// StandardPLC/Application/IO_CONFIG/INPUT_CONFIG_PI
PROGRAM INPUT_CONFIG_PI
VAR
	
	INPUT_A25: ifmFastInput.IncEncoder;
	CFDiag_INPUT_A25: ifmIOconfigDiagProt.ConfigDiagProt;
	INPUT_A26: ifmFastInput.IncEncoder;
	CFDiag_INPUT_A26: ifmIOconfigDiagProt.ConfigDiagProt;
	INPUT_A27: ifmFastInput.FastCount;
	CFDiag_INPUT_A27: ifmIOconfigDiagProt.ConfigDiagProt;
	INPUT_A28: ifmFastInput.FastCount;
	CFDiag_INPUT_A28: ifmIOconfigDiagProt.ConfigDiagProt;
	SET: ARRAY[0..70] OF SR;
	FastCount_0: ifmFastInput.FastCount;
	x1: BOOL;
	x2: REAL;
	x3: BOOL;
	x4: REAL;
END_VAR
VAR // added by the converter: edge detectors and wires of the graphical bodies
    _rt1, _rt2, _rt3, _rt4 : R_TRIG;
END_VAR

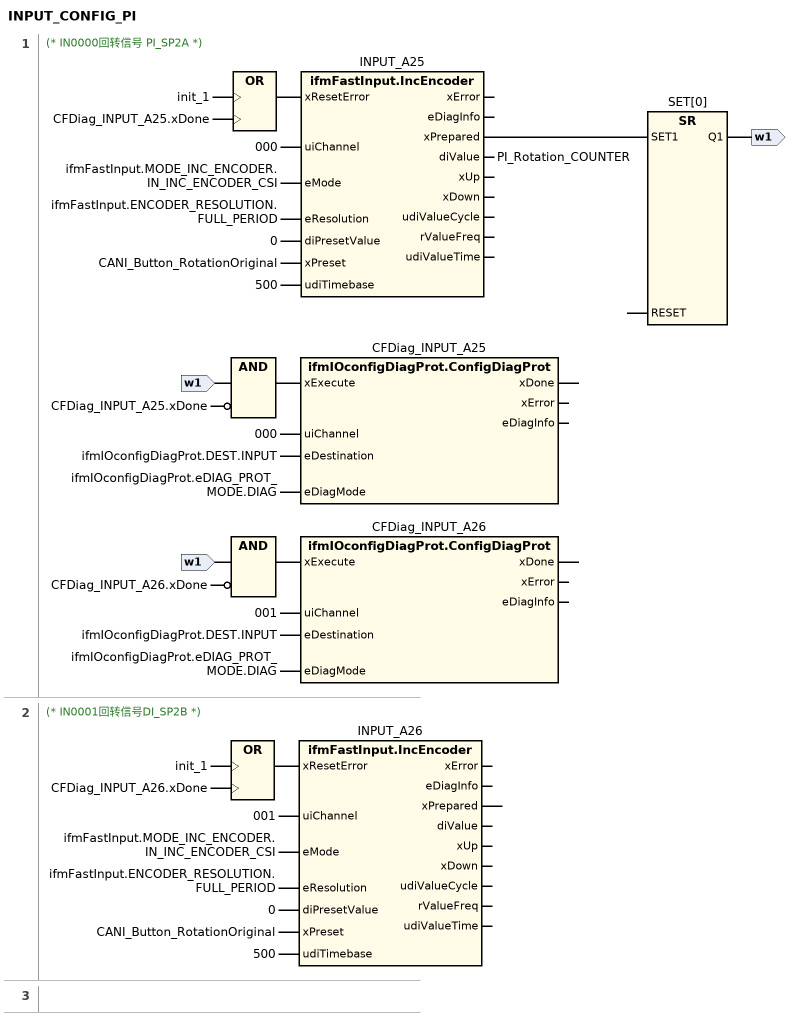
// NETWORK 1
//    (* IN0000回转信号 PI_SP2A *)
_rt1(CLK := init_1);
_rt2(CLK := CFDiag_INPUT_A25.xDone);
INPUT_A25(
    xResetError := _rt1.Q OR _rt2.Q,
    uiChannel := 000,
    eMode := ifmFastInput.MODE_INC_ENCODER.IN_INC_ENCODER_CSI,
    eResolution := ifmFastInput.ENCODER_RESOLUTION.FULL_PERIOD,
    diPresetValue := 0,
    xPreset := CANI_Button_RotationOriginal,
    udiTimebase := 500,
    diValue => PI_Rotation_COUNTER); // ifmFastInput.IncEncoder
SET[0](SET1 := INPUT_A25.xPrepared); // SR
CFDiag_INPUT_A25(
    xExecute := SET[0].Q1 AND NOT CFDiag_INPUT_A25.xDone,
    uiChannel := 000,
    eDestination := ifmIOconfigDiagProt.DEST.INPUT,
    eDiagMode := ifmIOconfigDiagProt.eDIAG_PROT_MODE.DIAG); // ifmIOconfigDiagProt.ConfigDiagProt
CFDiag_INPUT_A26(
    xExecute := SET[0].Q1 AND NOT CFDiag_INPUT_A26.xDone,
    uiChannel := 001,
    eDestination := ifmIOconfigDiagProt.DEST.INPUT,
    eDiagMode := ifmIOconfigDiagProt.eDIAG_PROT_MODE.DIAG); // ifmIOconfigDiagProt.ConfigDiagProt

// NETWORK 2
// (* IN0001回转信号DI_SP2B *)
_rt3(CLK := init_1);
_rt4(CLK := CFDiag_INPUT_A26.xDone);
INPUT_A26(
    xResetError := _rt3.Q OR _rt4.Q,
    uiChannel := 001,
    eMode := ifmFastInput.MODE_INC_ENCODER.IN_INC_ENCODER_CSI,
    eResolution := ifmFastInput.ENCODER_RESOLUTION.FULL_PERIOD,
    diPresetValue := 0,
    xPreset := CANI_Button_RotationOriginal,
    udiTimebase := 500); // ifmFastInput.IncEncoder

// NETWORK 3

END_PROGRAM

// StandardPLC/Application/IO_CONFIG/OUTPUT_CONFID
PROGRAM OUTPUT_CONFID
VAR
	SYSTEMSUPPLY:ifmIOcommon.SystemSupply;
	OUTGROUP0:ifmOutGroup.OutputGroup;
	OUTGROUP1:ifmOutGroup.OutputGroup;
	OUTGROUP2:ifmOutGroup.OutputGroup;
	OUTGROUP3:ifmOutGroup.OutputGroup;
	OUTGROUP4:ifmOutGroup.OutputGroup;
	OUTGROUP5:ifmOutGroup.OutputGroup;
(*******PWM*******)
	PWMI_A06: ifmOutPWM.CurrentControl;
//	PWMI_A06: ifmOutPWM.PWM1000;
	PWMI_A07: ifmOutPWM.PWM1000;
	PWMI_A08: ifmOutPWM.CurrentControl;
	PWMI_A09: ifmOutPWM.PWM1000;
	PWMI_A10: ifmOutPWM.CurrentControl;
	PWMI_A11: ifmOutPWM.PWM1000;
	PWMI_A12: ifmOutPWM.CurrentControl;
	PWMI_A13: ifmOutPWM.CurrentControl;
	PWMI_A14: ifmOutPWM.CurrentControl;
	PWMI_A16: ifmOutPWM.CurrentControl;
//	PWMI_A16: ifmOutPWM.PWM1000;
	PWMI_A17: ifmOutPWM.PWM1000;
	PWMI_A18: ifmOutPWM.CurrentControl;
//	PWMI_A18: CONTROL_OCC_CR7xxS;
	PWMI_A19: ifmOutPWM.PWM1000;
	PWMI_A20: ifmOutPWM.CurrentControl;
	PWMI_A21: ifmOutPWM.PWM1000;
	PWMI_A22: ifmOutPWM.CurrentControl;
	PWMI_A23: ifmOutPWM.CurrentControl;
	PWMI_A24: ifmOutPWM.CurrentControl;
	PWMI_A73: ifmOutPWM.CurrentControl;
	PWMI_A74: ifmOutPWM.PWM1000;
	PWMI_A75: ifmOutPWM.CurrentControl;
	PWMI_A76: ifmOutPWM.PWM1000;
	PWMI_A77: ifmOutPWM.CurrentControl;
	PWMI_A78: ifmOutPWM.PWM1000;
	PWMI_A79: ifmOutPWM.CurrentControl;
	PWMI_A80: ifmOutPWM.CurrentControl;
	PWMI_A81: ifmOutPWM.CurrentControl;
	
	PWMI_B16: ifmOutPWM.CurrentControl;
	PWMI_B17: ifmOutPWM.PWM1000;
	PWMI_B18: ifmOutPWM.CurrentControl;
	PWMI_B19: ifmOutPWM.PWM1000;
	PWMI_B20: ifmOutPWM.CurrentControl;
	PWMI_B21: ifmOutPWM.PWM1000;
	PWMI_B22: ifmOutPWM.CurrentControl;
	PWMI_B23: ifmOutPWM.CurrentControl;
	PWMI_B24: ifmOutPWM.CurrentControl;
	PWMI_B63: ifmOutPWM.CurrentControl;
	PWMI_B64: ifmOutPWM.PWM1000;
	PWMI_B65: ifmOutPWM.CurrentControl;
	PWMI_B66: ifmOutPWM.PWM1000;
	PWMI_B67: ifmOutPWM.CurrentControl;
//	PWMI_B68: ifmOutPWM.PWM1000;
	DOH_B68:ifmIOcommon.Output;
	DOH_B66:ifmIOcommon.Output;
	PWMI_B69: ifmOutPWM.CurrentControl;
	PWMI_B70: ifmOutPWM.CurrentControl;
	//PWMI_B71: ifmOutPWM.CurrentControl;
	DOH_B71:ifmIOcommon.Output;
	PWMI_B73: ifmOutPWM.CurrentControl;
	PWMI_B74: ifmOutPWM.PWM1000;
	PWMI_B75: ifmOutPWM.CurrentControl;
	//PWMI_B76: ifmOutPWM.PWM1000;
	DOH_B76:ifmIOcommon.Output;
	PWMI_B77: ifmOutPWM.CurrentControl;
	//PWMI_B78: ifmOutPWM.PWM1000;
	DOH_B78:ifmIOcommon.Output;
	PWMI_B79: ifmOutPWM.CurrentControl;
	PWMI_B80: ifmOutPWM.CurrentControl;
	PWMI_B81: ifmOutPWM.CurrentControl;
	//PWM参数
	diFre_i:UINT:=0;
	diVal_i:UINT:=0;
	KP:USINT:=50;
	KI:USINT:=50;
	StartRatio:UINT:=100;
	UI_Frequency:UINT:=160;
	r_ramp: INT:=1000;
	f_ramp: INT:=1000;
	TIMEbase: TIME:=T#200MS;
	BLINK_0: BLINK;
	vagroup_1: BOOL:=TRUE;
	
END_VAR

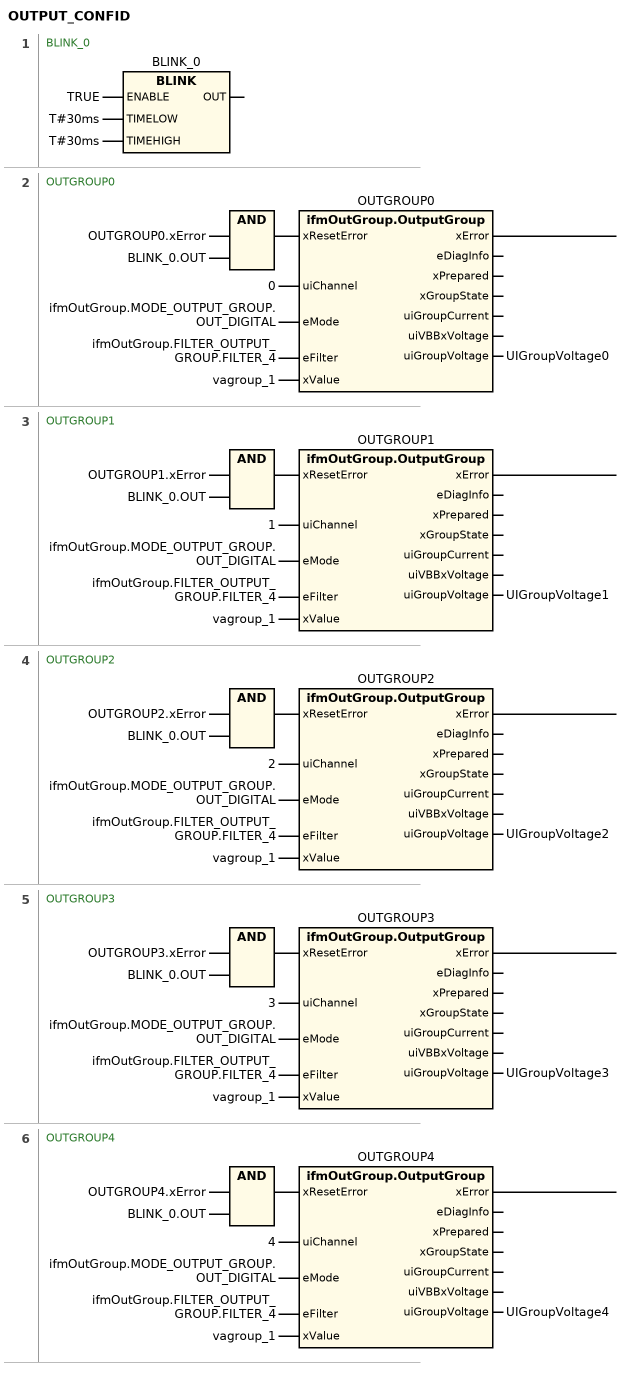
// NETWORK 1
// BLINK_0
BLINK_0(ENABLE := TRUE, TIMELOW := T#30ms, TIMEHIGH := T#30ms); // BLINK

// NETWORK 2
// OUTGROUP0
OUTGROUP0(
    xResetError := OUTGROUP0.xError AND BLINK_0.OUT,
    uiChannel := 0,
    eMode := ifmOutGroup.MODE_OUTPUT_GROUP.OUT_DIGITAL,
    eFilter := ifmOutGroup.FILTER_OUTPUT_GROUP.FILTER_4,
    xValue := vagroup_1,
    uiGroupVoltage => UIGroupVoltage0); // ifmOutGroup.OutputGroup

// NETWORK 3
// OUTGROUP1
OUTGROUP1(
    xResetError := OUTGROUP1.xError AND BLINK_0.OUT,
    uiChannel := 1,
    eMode := ifmOutGroup.MODE_OUTPUT_GROUP.OUT_DIGITAL,
    eFilter := ifmOutGroup.FILTER_OUTPUT_GROUP.FILTER_4,
    xValue := vagroup_1,
    uiGroupVoltage => UIGroupVoltage1); // ifmOutGroup.OutputGroup

// NETWORK 4
// OUTGROUP2
OUTGROUP2(
    xResetError := OUTGROUP2.xError AND BLINK_0.OUT,
    uiChannel := 2,
    eMode := ifmOutGroup.MODE_OUTPUT_GROUP.OUT_DIGITAL,
    eFilter := ifmOutGroup.FILTER_OUTPUT_GROUP.FILTER_4,
    xValue := vagroup_1,
    uiGroupVoltage => UIGroupVoltage2); // ifmOutGroup.OutputGroup

// NETWORK 5
// OUTGROUP3
OUTGROUP3(
    xResetError := OUTGROUP3.xError AND BLINK_0.OUT,
    uiChannel := 3,
    eMode := ifmOutGroup.MODE_OUTPUT_GROUP.OUT_DIGITAL,
    eFilter := ifmOutGroup.FILTER_OUTPUT_GROUP.FILTER_4,
    xValue := vagroup_1,
    uiGroupVoltage => UIGroupVoltage3); // ifmOutGroup.OutputGroup

// NETWORK 6
// OUTGROUP4
OUTGROUP4(
    xResetError := OUTGROUP4.xError AND BLINK_0.OUT,
    uiChannel := 4,
    eMode := ifmOutGroup.MODE_OUTPUT_GROUP.OUT_DIGITAL,
    eFilter := ifmOutGroup.FILTER_OUTPUT_GROUP.FILTER_4,
    xValue := vagroup_1,
    uiGroupVoltage => UIGroupVoltage4); // ifmOutGroup.OutputGroup

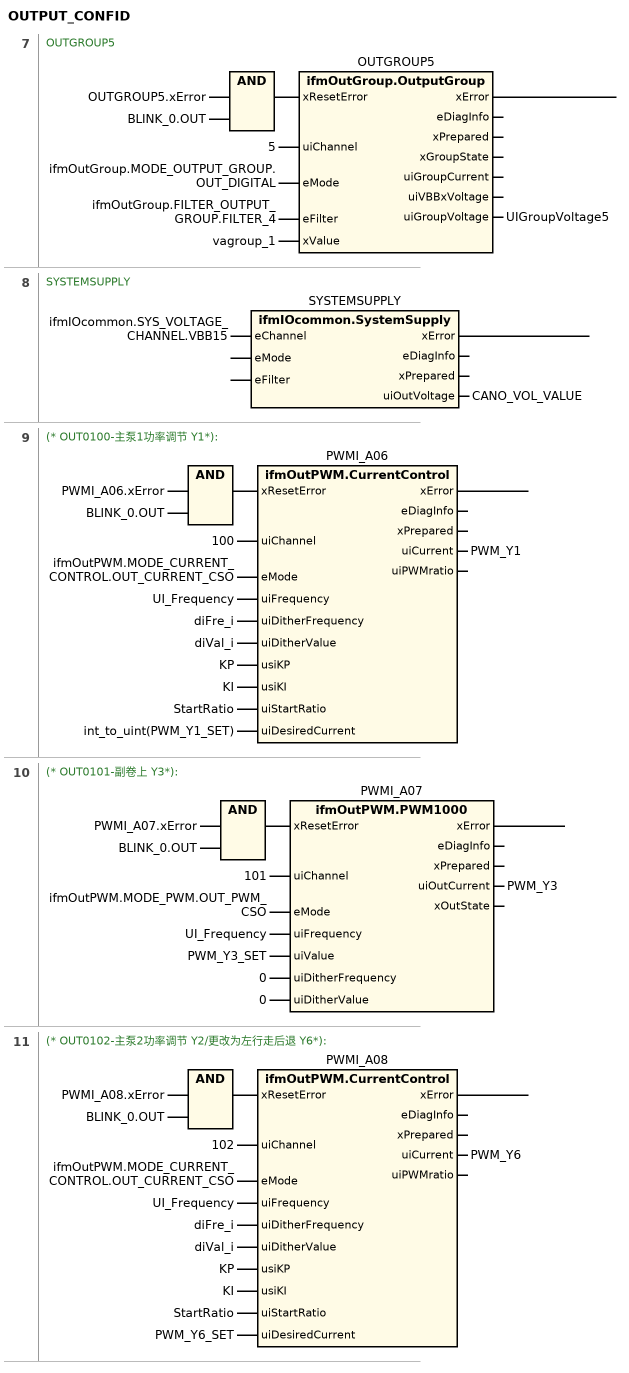
// NETWORK 7
// OUTGROUP5
OUTGROUP5(
    xResetError := OUTGROUP5.xError AND BLINK_0.OUT,
    uiChannel := 5,
    eMode := ifmOutGroup.MODE_OUTPUT_GROUP.OUT_DIGITAL,
    eFilter := ifmOutGroup.FILTER_OUTPUT_GROUP.FILTER_4,
    xValue := vagroup_1,
    uiGroupVoltage => UIGroupVoltage5); // ifmOutGroup.OutputGroup

// NETWORK 8
// SYSTEMSUPPLY
SYSTEMSUPPLY(eChannel := ifmIOcommon.SYS_VOLTAGE_CHANNEL.VBB15, uiOutVoltage => CANO_VOL_VALUE); // ifmIOcommon.SystemSupply

// NETWORK 9
// (* OUT0100-主泵1功率调节 Y1*):
PWMI_A06(
    xResetError := PWMI_A06.xError AND BLINK_0.OUT,
    uiChannel := 100,
    eMode := ifmOutPWM.MODE_CURRENT_CONTROL.OUT_CURRENT_CSO,
    uiFrequency := UI_Frequency,
    uiDitherFrequency := diFre_i,
    uiDitherValue := diVal_i,
    usiKP := KP,
    usiKI := KI,
    uiStartRatio := StartRatio,
    uiDesiredCurrent := int_to_uint(PWM_Y1_SET),
    uiCurrent => PWM_Y1); // ifmOutPWM.CurrentControl

// NETWORK 10
// (* OUT0101-副卷上 Y3*):
PWMI_A07(
    xResetError := PWMI_A07.xError AND BLINK_0.OUT,
    uiChannel := 101,
    eMode := ifmOutPWM.MODE_PWM.OUT_PWM_CSO,
    uiFrequency := UI_Frequency,
    uiValue := PWM_Y3_SET,
    uiDitherFrequency := 0,
    uiDitherValue := 0,
    uiOutCurrent => PWM_Y3); // ifmOutPWM.PWM1000

// NETWORK 11
// (* OUT0102-主泵2功率调节 Y2/更改为左行走后退 Y6*):
PWMI_A08(
    xResetError := PWMI_A08.xError AND BLINK_0.OUT,
    uiChannel := 102,
    eMode := ifmOutPWM.MODE_CURRENT_CONTROL.OUT_CURRENT_CSO,
    uiFrequency := UI_Frequency,
    uiDitherFrequency := diFre_i,
    uiDitherValue := diVal_i,
    usiKP := KP,
    usiKI := KI,
    uiStartRatio := StartRatio,
    uiDesiredCurrent := PWM_Y6_SET,
    uiCurrent => PWM_Y6); // ifmOutPWM.CurrentControl

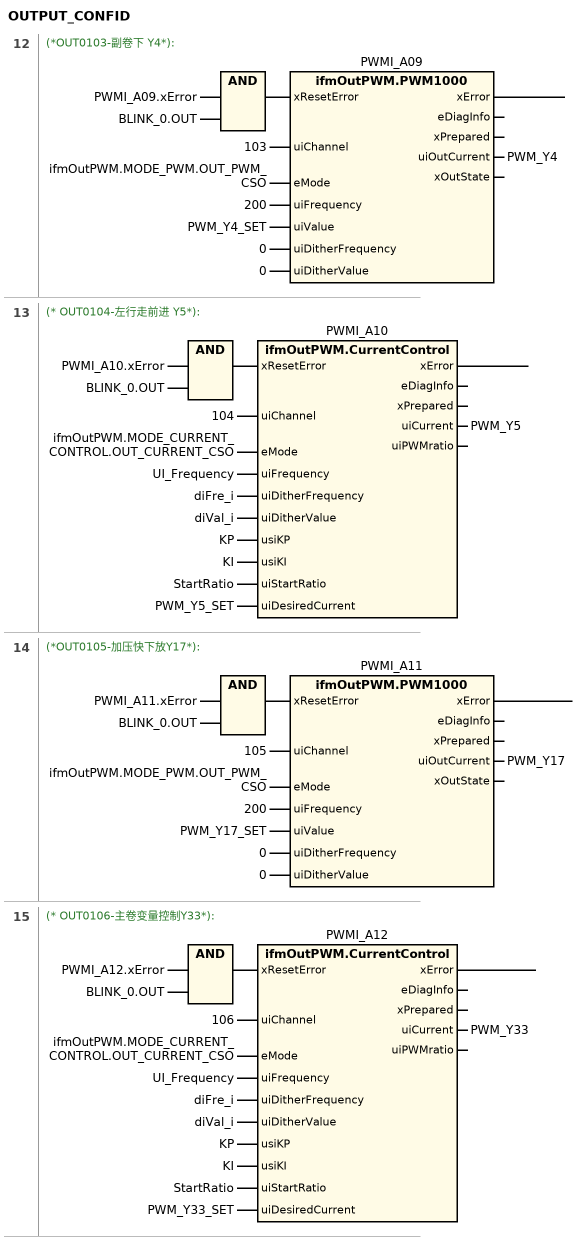
// NETWORK 12
// (*OUT0103-副卷下 Y4*):
PWMI_A09(
    xResetError := PWMI_A09.xError AND BLINK_0.OUT,
    uiChannel := 103,
    eMode := ifmOutPWM.MODE_PWM.OUT_PWM_CSO,
    uiFrequency := 200,
    uiValue := PWM_Y4_SET,
    uiDitherFrequency := 0,
    uiDitherValue := 0,
    uiOutCurrent => PWM_Y4); // ifmOutPWM.PWM1000

// NETWORK 13
// (* OUT0104-左行走前进 Y5*):
PWMI_A10(
    xResetError := PWMI_A10.xError AND BLINK_0.OUT,
    uiChannel := 104,
    eMode := ifmOutPWM.MODE_CURRENT_CONTROL.OUT_CURRENT_CSO,
    uiFrequency := UI_Frequency,
    uiDitherFrequency := diFre_i,
    uiDitherValue := diVal_i,
    usiKP := KP,
    usiKI := KI,
    uiStartRatio := StartRatio,
    uiDesiredCurrent := PWM_Y5_SET,
    uiCurrent => PWM_Y5); // ifmOutPWM.CurrentControl

// NETWORK 14
// (*OUT0105-加压快下放Y17*):
PWMI_A11(
    xResetError := PWMI_A11.xError AND BLINK_0.OUT,
    uiChannel := 105,
    eMode := ifmOutPWM.MODE_PWM.OUT_PWM_CSO,
    uiFrequency := 200,
    uiValue := PWM_Y17_SET,
    uiDitherFrequency := 0,
    uiDitherValue := 0,
    uiOutCurrent => PWM_Y17); // ifmOutPWM.PWM1000

// NETWORK 15
// (* OUT0106-主卷变量控制Y33*):
PWMI_A12(
    xResetError := PWMI_A12.xError AND BLINK_0.OUT,
    uiChannel := 106,
    eMode := ifmOutPWM.MODE_CURRENT_CONTROL.OUT_CURRENT_CSO,
    uiFrequency := UI_Frequency,
    uiDitherFrequency := diFre_i,
    uiDitherValue := diVal_i,
    usiKP := KP,
    usiKI := KI,
    uiStartRatio := StartRatio,
    uiDesiredCurrent := PWM_Y33_SET,
    uiCurrent => PWM_Y33); // ifmOutPWM.CurrentControl

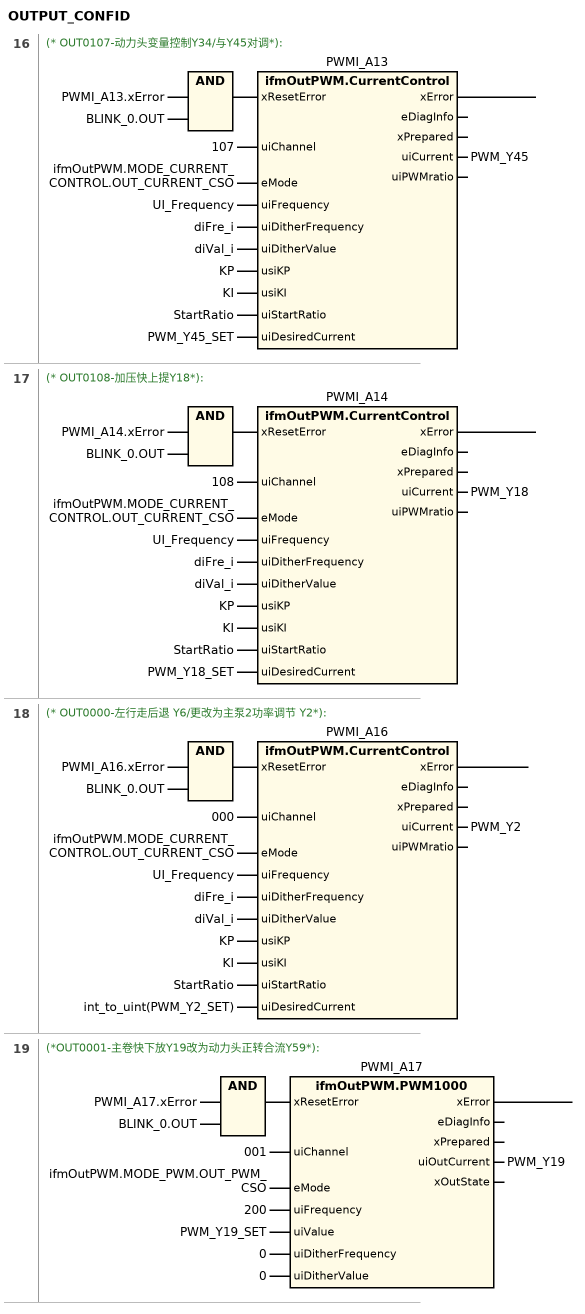
// NETWORK 16
// (* OUT0107-动力头变量控制Y34/与Y45对调*):
PWMI_A13(
    xResetError := PWMI_A13.xError AND BLINK_0.OUT,
    uiChannel := 107,
    eMode := ifmOutPWM.MODE_CURRENT_CONTROL.OUT_CURRENT_CSO,
    uiFrequency := UI_Frequency,
    uiDitherFrequency := diFre_i,
    uiDitherValue := diVal_i,
    usiKP := KP,
    usiKI := KI,
    uiStartRatio := StartRatio,
    uiDesiredCurrent := PWM_Y45_SET,
    uiCurrent => PWM_Y45); // ifmOutPWM.CurrentControl

// NETWORK 17
// (* OUT0108-加压快上提Y18*):
PWMI_A14(
    xResetError := PWMI_A14.xError AND BLINK_0.OUT,
    uiChannel := 108,
    eMode := ifmOutPWM.MODE_CURRENT_CONTROL.OUT_CURRENT_CSO,
    uiFrequency := UI_Frequency,
    uiDitherFrequency := diFre_i,
    uiDitherValue := diVal_i,
    usiKP := KP,
    usiKI := KI,
    uiStartRatio := StartRatio,
    uiDesiredCurrent := PWM_Y18_SET,
    uiCurrent => PWM_Y18); // ifmOutPWM.CurrentControl

// NETWORK 18
// (* OUT0000-左行走后退 Y6/更改为主泵2功率调节 Y2*):
PWMI_A16(
    xResetError := PWMI_A16.xError AND BLINK_0.OUT,
    uiChannel := 000,
    eMode := ifmOutPWM.MODE_CURRENT_CONTROL.OUT_CURRENT_CSO,
    uiFrequency := UI_Frequency,
    uiDitherFrequency := diFre_i,
    uiDitherValue := diVal_i,
    usiKP := KP,
    usiKI := KI,
    uiStartRatio := StartRatio,
    uiDesiredCurrent := int_to_uint(PWM_Y2_SET),
    uiCurrent => PWM_Y2); // ifmOutPWM.CurrentControl

// NETWORK 19
// (*OUT0001-主卷快下放Y19改为动力头正转合流Y59*):
PWMI_A17(
    xResetError := PWMI_A17.xError AND BLINK_0.OUT,
    uiChannel := 001,
    eMode := ifmOutPWM.MODE_PWM.OUT_PWM_CSO,
    uiFrequency := 200,
    uiValue := PWM_Y19_SET,
    uiDitherFrequency := 0,
    uiDitherValue := 0,
    uiOutCurrent => PWM_Y19); // ifmOutPWM.PWM1000

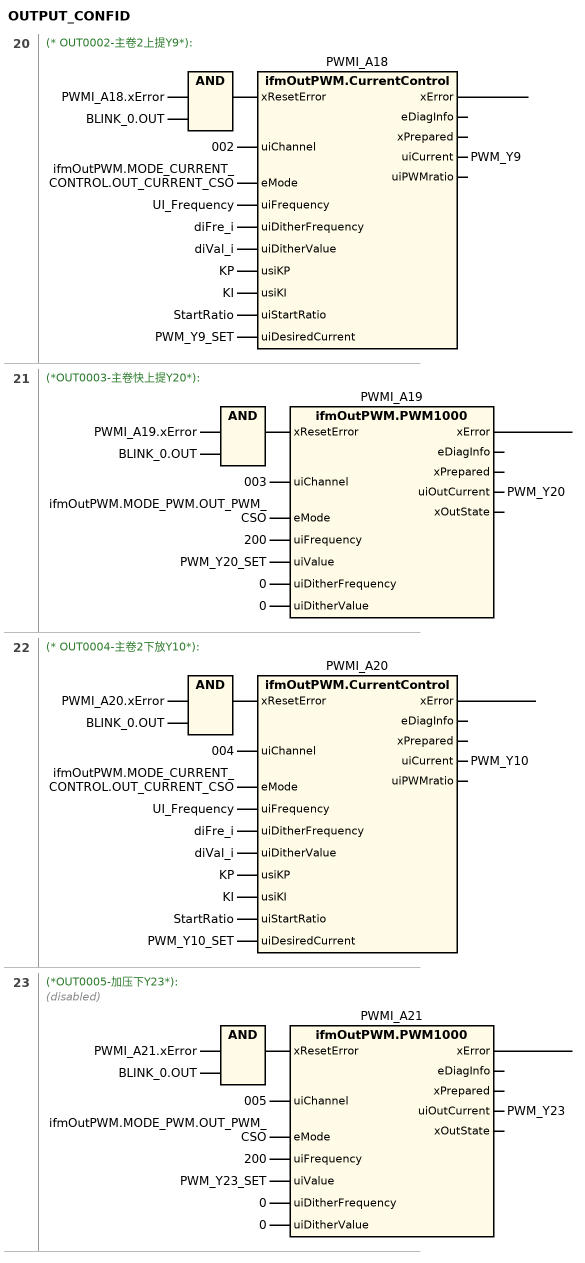
// NETWORK 20
// (* OUT0002-主卷2上提Y9*):
PWMI_A18(
    xResetError := PWMI_A18.xError AND BLINK_0.OUT,
    uiChannel := 002,
    eMode := ifmOutPWM.MODE_CURRENT_CONTROL.OUT_CURRENT_CSO,
    uiFrequency := UI_Frequency,
    uiDitherFrequency := diFre_i,
    uiDitherValue := diVal_i,
    usiKP := KP,
    usiKI := KI,
    uiStartRatio := StartRatio,
    uiDesiredCurrent := PWM_Y9_SET,
    uiCurrent => PWM_Y9); // ifmOutPWM.CurrentControl

// NETWORK 21
// (*OUT0003-主卷快上提Y20*):
PWMI_A19(
    xResetError := PWMI_A19.xError AND BLINK_0.OUT,
    uiChannel := 003,
    eMode := ifmOutPWM.MODE_PWM.OUT_PWM_CSO,
    uiFrequency := 200,
    uiValue := PWM_Y20_SET,
    uiDitherFrequency := 0,
    uiDitherValue := 0,
    uiOutCurrent => PWM_Y20); // ifmOutPWM.PWM1000

// NETWORK 22
// (* OUT0004-主卷2下放Y10*):
PWMI_A20(
    xResetError := PWMI_A20.xError AND BLINK_0.OUT,
    uiChannel := 004,
    eMode := ifmOutPWM.MODE_CURRENT_CONTROL.OUT_CURRENT_CSO,
    uiFrequency := UI_Frequency,
    uiDitherFrequency := diFre_i,
    uiDitherValue := diVal_i,
    usiKP := KP,
    usiKI := KI,
    uiStartRatio := StartRatio,
    uiDesiredCurrent := PWM_Y10_SET,
    uiCurrent => PWM_Y10); // ifmOutPWM.CurrentControl

// NETWORK 23 (disabled)
// (*OUT0005-加压下Y23*):
// PWMI_A21(
//     xResetError := PWMI_A21.xError AND BLINK_0.OUT,
//     uiChannel := 005,
//     eMode := ifmOutPWM.MODE_PWM.OUT_PWM_CSO,
//     uiFrequency := 200,
//     uiValue := PWM_Y23_SET,
//     uiDitherFrequency := 0,
//     uiDitherValue := 0,
//     uiOutCurrent => PWM_Y23); // ifmOutPWM.PWM1000

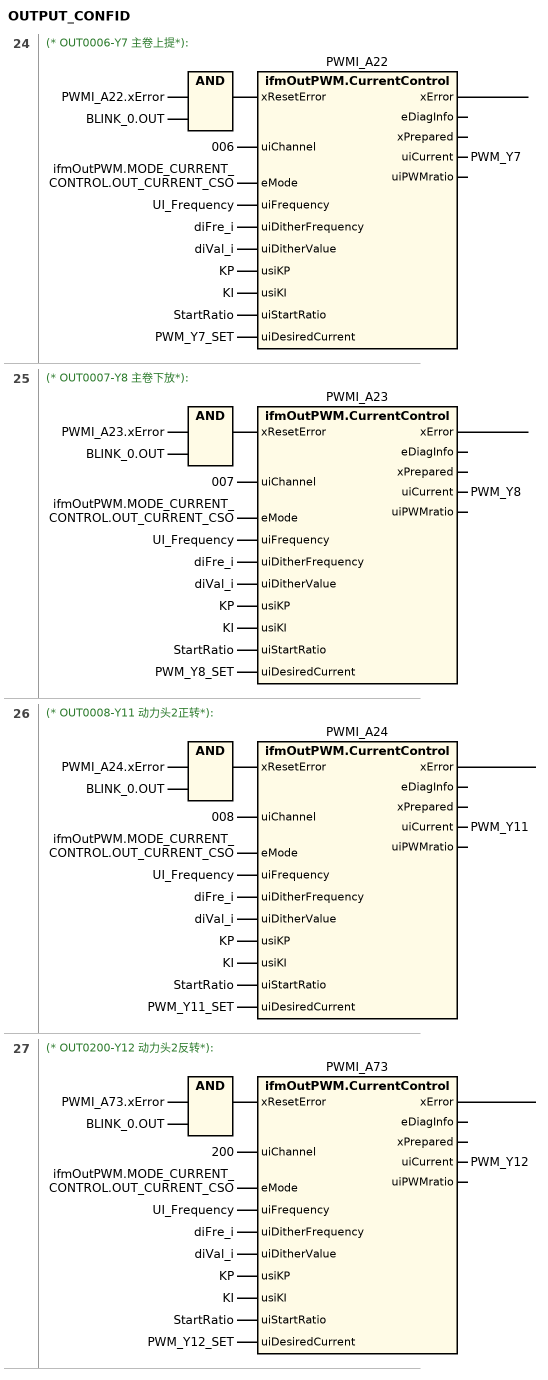
// NETWORK 24
// (* OUT0006-Y7 主卷上提*):
PWMI_A22(
    xResetError := PWMI_A22.xError AND BLINK_0.OUT,
    uiChannel := 006,
    eMode := ifmOutPWM.MODE_CURRENT_CONTROL.OUT_CURRENT_CSO,
    uiFrequency := UI_Frequency,
    uiDitherFrequency := diFre_i,
    uiDitherValue := diVal_i,
    usiKP := KP,
    usiKI := KI,
    uiStartRatio := StartRatio,
    uiDesiredCurrent := PWM_Y7_SET,
    uiCurrent => PWM_Y7); // ifmOutPWM.CurrentControl

// NETWORK 25
// (* OUT0007-Y8 主卷下放*):
PWMI_A23(
    xResetError := PWMI_A23.xError AND BLINK_0.OUT,
    uiChannel := 007,
    eMode := ifmOutPWM.MODE_CURRENT_CONTROL.OUT_CURRENT_CSO,
    uiFrequency := UI_Frequency,
    uiDitherFrequency := diFre_i,
    uiDitherValue := diVal_i,
    usiKP := KP,
    usiKI := KI,
    uiStartRatio := StartRatio,
    uiDesiredCurrent := PWM_Y8_SET,
    uiCurrent => PWM_Y8); // ifmOutPWM.CurrentControl

// NETWORK 26
// (* OUT0008-Y11 动力头2正转*):
PWMI_A24(
    xResetError := PWMI_A24.xError AND BLINK_0.OUT,
    uiChannel := 008,
    eMode := ifmOutPWM.MODE_CURRENT_CONTROL.OUT_CURRENT_CSO,
    uiFrequency := UI_Frequency,
    uiDitherFrequency := diFre_i,
    uiDitherValue := diVal_i,
    usiKP := KP,
    usiKI := KI,
    uiStartRatio := StartRatio,
    uiDesiredCurrent := PWM_Y11_SET,
    uiCurrent => PWM_Y11); // ifmOutPWM.CurrentControl

// NETWORK 27
// (* OUT0200-Y12 动力头2反转*):
PWMI_A73(
    xResetError := PWMI_A73.xError AND BLINK_0.OUT,
    uiChannel := 200,
    eMode := ifmOutPWM.MODE_CURRENT_CONTROL.OUT_CURRENT_CSO,
    uiFrequency := UI_Frequency,
    uiDitherFrequency := diFre_i,
    uiDitherValue := diVal_i,
    usiKP := KP,
    usiKI := KI,
    uiStartRatio := StartRatio,
    uiDesiredCurrent := PWM_Y12_SET,
    uiCurrent => PWM_Y12); // ifmOutPWM.CurrentControl

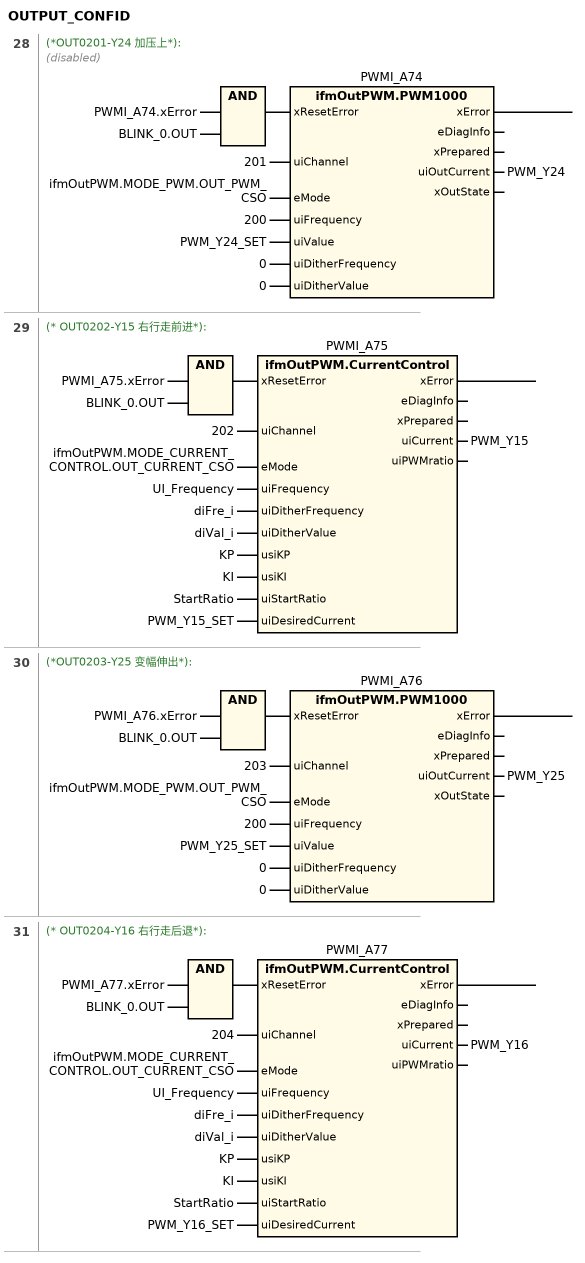
// NETWORK 28 (disabled)
// (*OUT0201-Y24 加压上*):
// PWMI_A74(
//     xResetError := PWMI_A74.xError AND BLINK_0.OUT,
//     uiChannel := 201,
//     eMode := ifmOutPWM.MODE_PWM.OUT_PWM_CSO,
//     uiFrequency := 200,
//     uiValue := PWM_Y24_SET,
//     uiDitherFrequency := 0,
//     uiDitherValue := 0,
//     uiOutCurrent => PWM_Y24); // ifmOutPWM.PWM1000

// NETWORK 29
// (* OUT0202-Y15 右行走前进*):
PWMI_A75(
    xResetError := PWMI_A75.xError AND BLINK_0.OUT,
    uiChannel := 202,
    eMode := ifmOutPWM.MODE_CURRENT_CONTROL.OUT_CURRENT_CSO,
    uiFrequency := UI_Frequency,
    uiDitherFrequency := diFre_i,
    uiDitherValue := diVal_i,
    usiKP := KP,
    usiKI := KI,
    uiStartRatio := StartRatio,
    uiDesiredCurrent := PWM_Y15_SET,
    uiCurrent => PWM_Y15); // ifmOutPWM.CurrentControl

// NETWORK 30
// (*OUT0203-Y25 变幅伸出*):
PWMI_A76(
    xResetError := PWMI_A76.xError AND BLINK_0.OUT,
    uiChannel := 203,
    eMode := ifmOutPWM.MODE_PWM.OUT_PWM_CSO,
    uiFrequency := 200,
    uiValue := PWM_Y25_SET,
    uiDitherFrequency := 0,
    uiDitherValue := 0,
    uiOutCurrent => PWM_Y25); // ifmOutPWM.PWM1000

// NETWORK 31
// (* OUT0204-Y16 右行走后退*):
PWMI_A77(
    xResetError := PWMI_A77.xError AND BLINK_0.OUT,
    uiChannel := 204,
    eMode := ifmOutPWM.MODE_CURRENT_CONTROL.OUT_CURRENT_CSO,
    uiFrequency := UI_Frequency,
    uiDitherFrequency := diFre_i,
    uiDitherValue := diVal_i,
    usiKP := KP,
    usiKI := KI,
    uiStartRatio := StartRatio,
    uiDesiredCurrent := PWM_Y16_SET,
    uiCurrent => PWM_Y16); // ifmOutPWM.CurrentControl

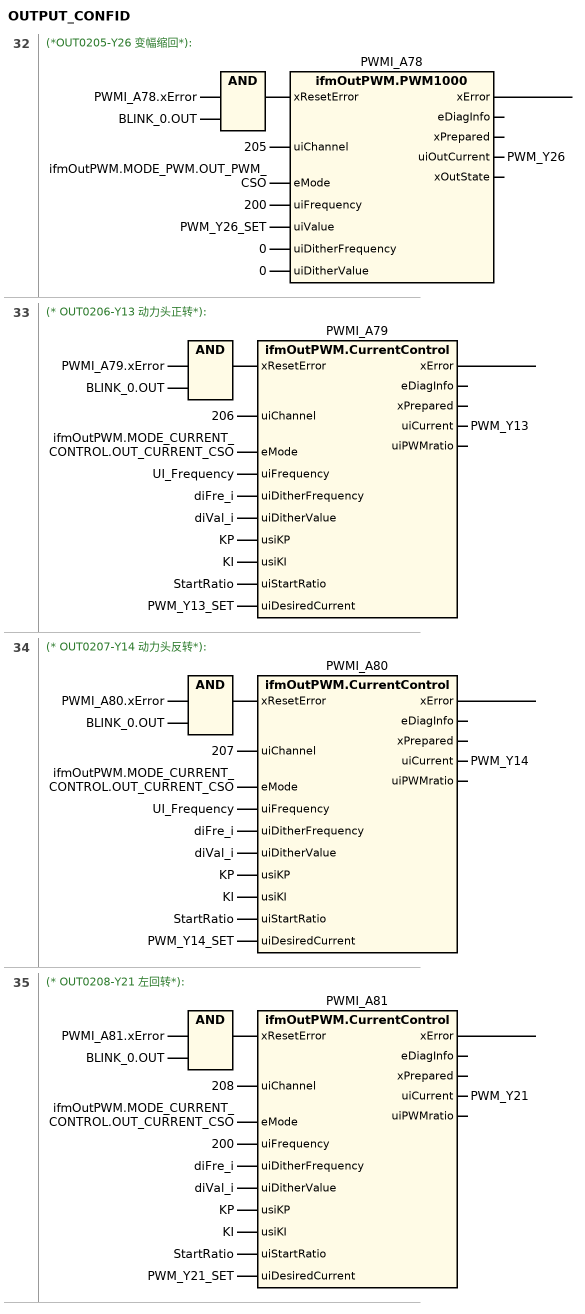
// NETWORK 32
// (*OUT0205-Y26 变幅缩回*):
PWMI_A78(
    xResetError := PWMI_A78.xError AND BLINK_0.OUT,
    uiChannel := 205,
    eMode := ifmOutPWM.MODE_PWM.OUT_PWM_CSO,
    uiFrequency := 200,
    uiValue := PWM_Y26_SET,
    uiDitherFrequency := 0,
    uiDitherValue := 0,
    uiOutCurrent => PWM_Y26); // ifmOutPWM.PWM1000

// NETWORK 33
// (* OUT0206-Y13 动力头正转*):
PWMI_A79(
    xResetError := PWMI_A79.xError AND BLINK_0.OUT,
    uiChannel := 206,
    eMode := ifmOutPWM.MODE_CURRENT_CONTROL.OUT_CURRENT_CSO,
    uiFrequency := UI_Frequency,
    uiDitherFrequency := diFre_i,
    uiDitherValue := diVal_i,
    usiKP := KP,
    usiKI := KI,
    uiStartRatio := StartRatio,
    uiDesiredCurrent := PWM_Y13_SET,
    uiCurrent => PWM_Y13); // ifmOutPWM.CurrentControl

// NETWORK 34
// (* OUT0207-Y14 动力头反转*):
PWMI_A80(
    xResetError := PWMI_A80.xError AND BLINK_0.OUT,
    uiChannel := 207,
    eMode := ifmOutPWM.MODE_CURRENT_CONTROL.OUT_CURRENT_CSO,
    uiFrequency := UI_Frequency,
    uiDitherFrequency := diFre_i,
    uiDitherValue := diVal_i,
    usiKP := KP,
    usiKI := KI,
    uiStartRatio := StartRatio,
    uiDesiredCurrent := PWM_Y14_SET,
    uiCurrent => PWM_Y14); // ifmOutPWM.CurrentControl

// NETWORK 35
// (* OUT0208-Y21 左回转*):
PWMI_A81(
    xResetError := PWMI_A81.xError AND BLINK_0.OUT,
    uiChannel := 208,
    eMode := ifmOutPWM.MODE_CURRENT_CONTROL.OUT_CURRENT_CSO,
    uiFrequency := 200,
    uiDitherFrequency := diFre_i,
    uiDitherValue := diVal_i,
    usiKP := KP,
    usiKI := KI,
    uiStartRatio := StartRatio,
    uiDesiredCurrent := PWM_Y21_SET,
    uiCurrent => PWM_Y21); // ifmOutPWM.CurrentControl

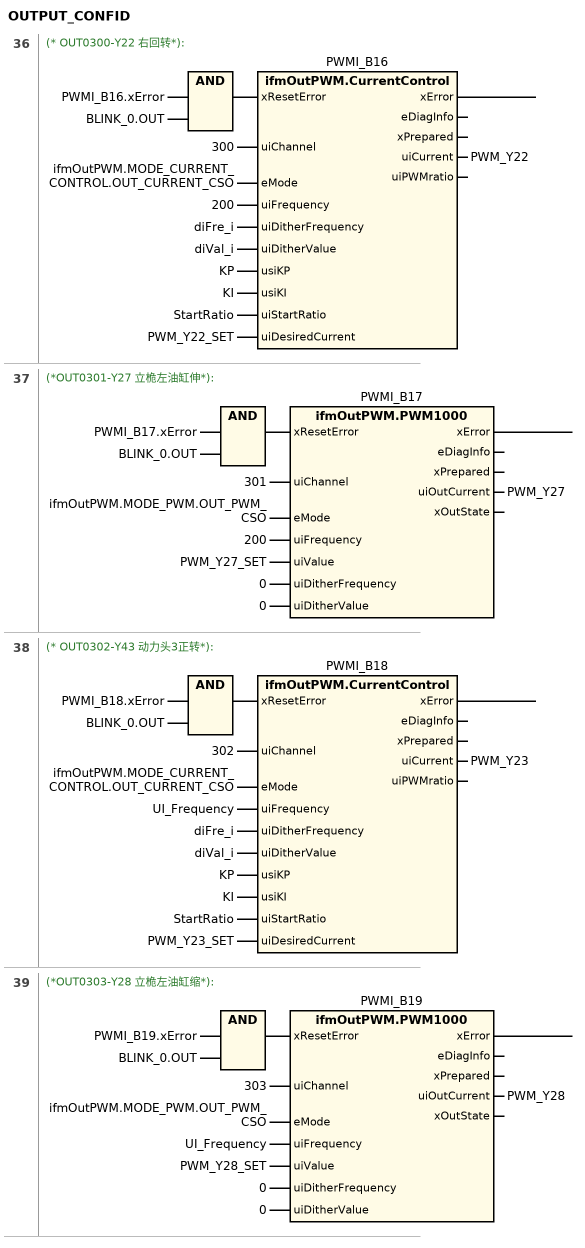
// NETWORK 36
// (* OUT0300-Y22 右回转*):
PWMI_B16(
    xResetError := PWMI_B16.xError AND BLINK_0.OUT,
    uiChannel := 300,
    eMode := ifmOutPWM.MODE_CURRENT_CONTROL.OUT_CURRENT_CSO,
    uiFrequency := 200,
    uiDitherFrequency := diFre_i,
    uiDitherValue := diVal_i,
    usiKP := KP,
    usiKI := KI,
    uiStartRatio := StartRatio,
    uiDesiredCurrent := PWM_Y22_SET,
    uiCurrent => PWM_Y22); // ifmOutPWM.CurrentControl

// NETWORK 37
// (*OUT0301-Y27 立桅左油缸伸*):
PWMI_B17(
    xResetError := PWMI_B17.xError AND BLINK_0.OUT,
    uiChannel := 301,
    eMode := ifmOutPWM.MODE_PWM.OUT_PWM_CSO,
    uiFrequency := 200,
    uiValue := PWM_Y27_SET,
    uiDitherFrequency := 0,
    uiDitherValue := 0,
    uiOutCurrent => PWM_Y27); // ifmOutPWM.PWM1000

// NETWORK 38
// (* OUT0302-Y43 动力头3正转*):
PWMI_B18(
    xResetError := PWMI_B18.xError AND BLINK_0.OUT,
    uiChannel := 302,
    eMode := ifmOutPWM.MODE_CURRENT_CONTROL.OUT_CURRENT_CSO,
    uiFrequency := UI_Frequency,
    uiDitherFrequency := diFre_i,
    uiDitherValue := diVal_i,
    usiKP := KP,
    usiKI := KI,
    uiStartRatio := StartRatio,
    uiDesiredCurrent := PWM_Y23_SET,
    uiCurrent => PWM_Y23); // ifmOutPWM.CurrentControl

// NETWORK 39
// (*OUT0303-Y28 立桅左油缸缩*):
PWMI_B19(
    xResetError := PWMI_B19.xError AND BLINK_0.OUT,
    uiChannel := 303,
    eMode := ifmOutPWM.MODE_PWM.OUT_PWM_CSO,
    uiFrequency := UI_Frequency,
    uiValue := PWM_Y28_SET,
    uiDitherFrequency := 0,
    uiDitherValue := 0,
    uiOutCurrent => PWM_Y28); // ifmOutPWM.PWM1000

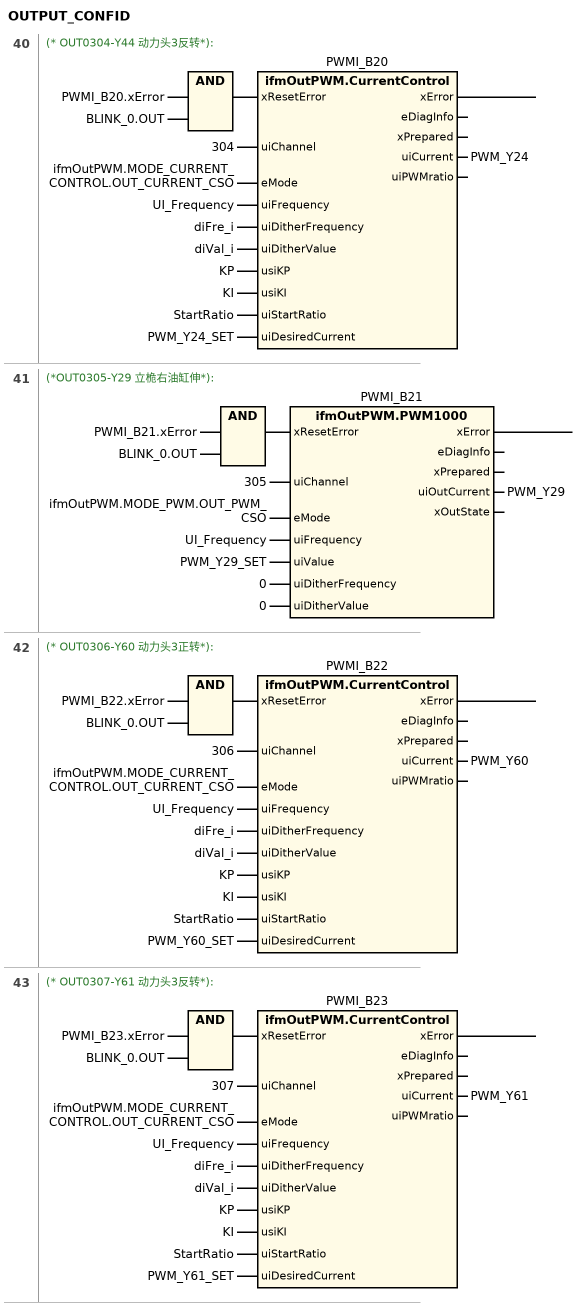
// NETWORK 40
// (* OUT0304-Y44 动力头3反转*):
PWMI_B20(
    xResetError := PWMI_B20.xError AND BLINK_0.OUT,
    uiChannel := 304,
    eMode := ifmOutPWM.MODE_CURRENT_CONTROL.OUT_CURRENT_CSO,
    uiFrequency := UI_Frequency,
    uiDitherFrequency := diFre_i,
    uiDitherValue := diVal_i,
    usiKP := KP,
    usiKI := KI,
    uiStartRatio := StartRatio,
    uiDesiredCurrent := PWM_Y24_SET,
    uiCurrent => PWM_Y24); // ifmOutPWM.CurrentControl

// NETWORK 41
// (*OUT0305-Y29 立桅右油缸伸*):
PWMI_B21(
    xResetError := PWMI_B21.xError AND BLINK_0.OUT,
    uiChannel := 305,
    eMode := ifmOutPWM.MODE_PWM.OUT_PWM_CSO,
    uiFrequency := UI_Frequency,
    uiValue := PWM_Y29_SET,
    uiDitherFrequency := 0,
    uiDitherValue := 0,
    uiOutCurrent => PWM_Y29); // ifmOutPWM.PWM1000

// NETWORK 42
// (* OUT0306-Y60 动力头3正转*):
PWMI_B22(
    xResetError := PWMI_B22.xError AND BLINK_0.OUT,
    uiChannel := 306,
    eMode := ifmOutPWM.MODE_CURRENT_CONTROL.OUT_CURRENT_CSO,
    uiFrequency := UI_Frequency,
    uiDitherFrequency := diFre_i,
    uiDitherValue := diVal_i,
    usiKP := KP,
    usiKI := KI,
    uiStartRatio := StartRatio,
    uiDesiredCurrent := PWM_Y60_SET,
    uiCurrent => PWM_Y60); // ifmOutPWM.CurrentControl

// NETWORK 43
// (* OUT0307-Y61 动力头3反转*):
PWMI_B23(
    xResetError := PWMI_B23.xError AND BLINK_0.OUT,
    uiChannel := 307,
    eMode := ifmOutPWM.MODE_CURRENT_CONTROL.OUT_CURRENT_CSO,
    uiFrequency := UI_Frequency,
    uiDitherFrequency := diFre_i,
    uiDitherValue := diVal_i,
    usiKP := KP,
    usiKI := KI,
    uiStartRatio := StartRatio,
    uiDesiredCurrent := PWM_Y61_SET,
    uiCurrent => PWM_Y61); // ifmOutPWM.CurrentControl

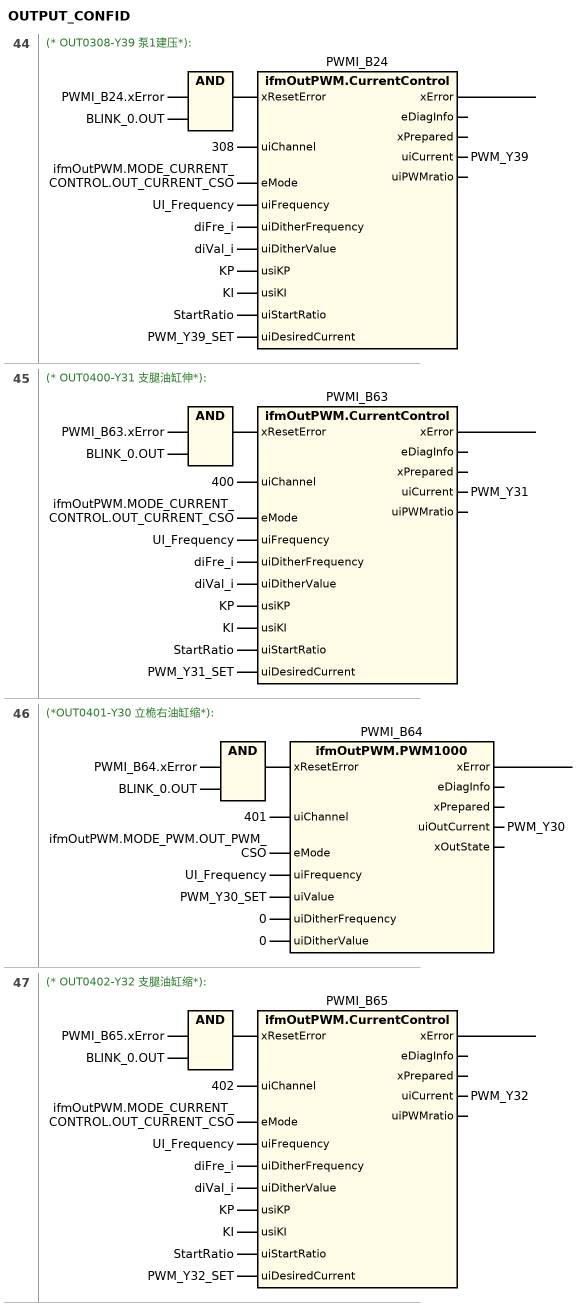
// NETWORK 44
// (* OUT0308-Y39 泵1建压*):
PWMI_B24(
    xResetError := PWMI_B24.xError AND BLINK_0.OUT,
    uiChannel := 308,
    eMode := ifmOutPWM.MODE_CURRENT_CONTROL.OUT_CURRENT_CSO,
    uiFrequency := UI_Frequency,
    uiDitherFrequency := diFre_i,
    uiDitherValue := diVal_i,
    usiKP := KP,
    usiKI := KI,
    uiStartRatio := StartRatio,
    uiDesiredCurrent := PWM_Y39_SET,
    uiCurrent => PWM_Y39); // ifmOutPWM.CurrentControl

// NETWORK 45
// (* OUT0400-Y31 支腿油缸伸*):
PWMI_B63(
    xResetError := PWMI_B63.xError AND BLINK_0.OUT,
    uiChannel := 400,
    eMode := ifmOutPWM.MODE_CURRENT_CONTROL.OUT_CURRENT_CSO,
    uiFrequency := UI_Frequency,
    uiDitherFrequency := diFre_i,
    uiDitherValue := diVal_i,
    usiKP := KP,
    usiKI := KI,
    uiStartRatio := StartRatio,
    uiDesiredCurrent := PWM_Y31_SET,
    uiCurrent => PWM_Y31); // ifmOutPWM.CurrentControl

// NETWORK 46
// (*OUT0401-Y30 立桅右油缸缩*):
PWMI_B64(
    xResetError := PWMI_B64.xError AND BLINK_0.OUT,
    uiChannel := 401,
    eMode := ifmOutPWM.MODE_PWM.OUT_PWM_CSO,
    uiFrequency := UI_Frequency,
    uiValue := PWM_Y30_SET,
    uiDitherFrequency := 0,
    uiDitherValue := 0,
    uiOutCurrent => PWM_Y30); // ifmOutPWM.PWM1000

// NETWORK 47
// (* OUT0402-Y32 支腿油缸缩*):
PWMI_B65(
    xResetError := PWMI_B65.xError AND BLINK_0.OUT,
    uiChannel := 402,
    eMode := ifmOutPWM.MODE_CURRENT_CONTROL.OUT_CURRENT_CSO,
    uiFrequency := UI_Frequency,
    uiDitherFrequency := diFre_i,
    uiDitherValue := diVal_i,
    usiKP := KP,
    usiKI := KI,
    uiStartRatio := StartRatio,
    uiDesiredCurrent := PWM_Y32_SET,
    uiCurrent => PWM_Y32); // ifmOutPWM.CurrentControl

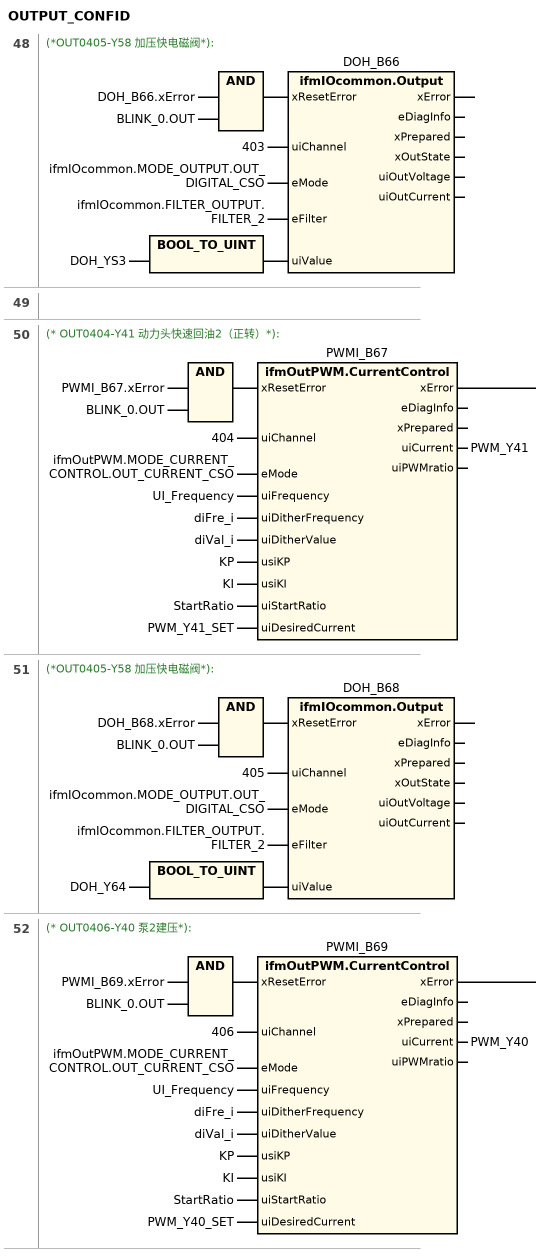
// NETWORK 48
// (*OUT0405-Y58 加压快电磁阀*):
DOH_B66(
    xResetError := DOH_B66.xError AND BLINK_0.OUT,
    uiChannel := 403,
    eMode := ifmIOcommon.MODE_OUTPUT.OUT_DIGITAL_CSO,
    eFilter := ifmIOcommon.FILTER_OUTPUT.FILTER_2,
    uiValue := BOOL_TO_UINT(DOH_YS3)); // ifmIOcommon.Output

// NETWORK 49

// NETWORK 50
// (* OUT0404-Y41 动力头快速回油2（正转）*):
PWMI_B67(
    xResetError := PWMI_B67.xError AND BLINK_0.OUT,
    uiChannel := 404,
    eMode := ifmOutPWM.MODE_CURRENT_CONTROL.OUT_CURRENT_CSO,
    uiFrequency := UI_Frequency,
    uiDitherFrequency := diFre_i,
    uiDitherValue := diVal_i,
    usiKP := KP,
    usiKI := KI,
    uiStartRatio := StartRatio,
    uiDesiredCurrent := PWM_Y41_SET,
    uiCurrent => PWM_Y41); // ifmOutPWM.CurrentControl

// NETWORK 51
// (*OUT0405-Y58 加压快电磁阀*):
DOH_B68(
    xResetError := DOH_B68.xError AND BLINK_0.OUT,
    uiChannel := 405,
    eMode := ifmIOcommon.MODE_OUTPUT.OUT_DIGITAL_CSO,
    eFilter := ifmIOcommon.FILTER_OUTPUT.FILTER_2,
    uiValue := BOOL_TO_UINT(DOH_Y64)); // ifmIOcommon.Output

// NETWORK 52
// (* OUT0406-Y40 泵2建压*):
PWMI_B69(
    xResetError := PWMI_B69.xError AND BLINK_0.OUT,
    uiChannel := 406,
    eMode := ifmOutPWM.MODE_CURRENT_CONTROL.OUT_CURRENT_CSO,
    uiFrequency := UI_Frequency,
    uiDitherFrequency := diFre_i,
    uiDitherValue := diVal_i,
    usiKP := KP,
    usiKI := KI,
    uiStartRatio := StartRatio,
    uiDesiredCurrent := PWM_Y40_SET,
    uiCurrent => PWM_Y40); // ifmOutPWM.CurrentControl

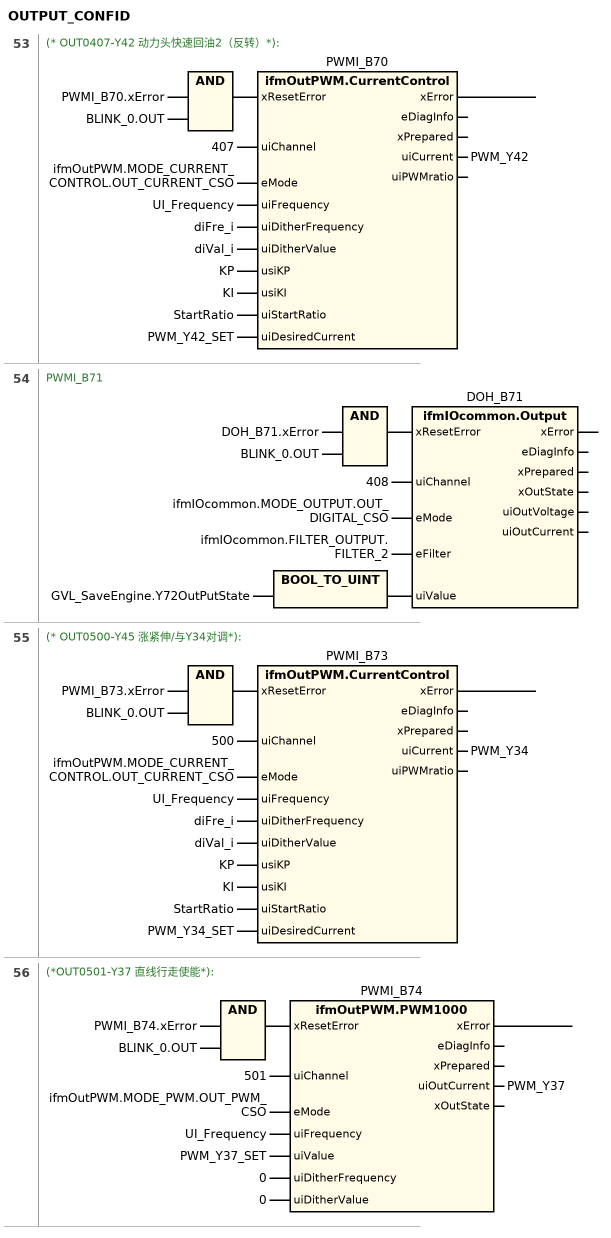
// NETWORK 53
// (* OUT0407-Y42 动力头快速回油2（反转）*):
PWMI_B70(
    xResetError := PWMI_B70.xError AND BLINK_0.OUT,
    uiChannel := 407,
    eMode := ifmOutPWM.MODE_CURRENT_CONTROL.OUT_CURRENT_CSO,
    uiFrequency := UI_Frequency,
    uiDitherFrequency := diFre_i,
    uiDitherValue := diVal_i,
    usiKP := KP,
    usiKI := KI,
    uiStartRatio := StartRatio,
    uiDesiredCurrent := PWM_Y42_SET,
    uiCurrent => PWM_Y42); // ifmOutPWM.CurrentControl

// NETWORK 54
// PWMI_B71
DOH_B71(
    xResetError := DOH_B71.xError AND BLINK_0.OUT,
    uiChannel := 408,
    eMode := ifmIOcommon.MODE_OUTPUT.OUT_DIGITAL_CSO,
    eFilter := ifmIOcommon.FILTER_OUTPUT.FILTER_2,
    uiValue := BOOL_TO_UINT(GVL_SaveEngine.Y72OutPutState)); // ifmIOcommon.Output

// NETWORK 55
// (* OUT0500-Y45 涨紧伸/与Y34对调*):
PWMI_B73(
    xResetError := PWMI_B73.xError AND BLINK_0.OUT,
    uiChannel := 500,
    eMode := ifmOutPWM.MODE_CURRENT_CONTROL.OUT_CURRENT_CSO,
    uiFrequency := UI_Frequency,
    uiDitherFrequency := diFre_i,
    uiDitherValue := diVal_i,
    usiKP := KP,
    usiKI := KI,
    uiStartRatio := StartRatio,
    uiDesiredCurrent := PWM_Y34_SET,
    uiCurrent => PWM_Y34); // ifmOutPWM.CurrentControl

// NETWORK 56
// (*OUT0501-Y37 直线行走使能*):
PWMI_B74(
    xResetError := PWMI_B74.xError AND BLINK_0.OUT,
    uiChannel := 501,
    eMode := ifmOutPWM.MODE_PWM.OUT_PWM_CSO,
    uiFrequency := UI_Frequency,
    uiValue := PWM_Y37_SET,
    uiDitherFrequency := 0,
    uiDitherValue := 0,
    uiOutCurrent => PWM_Y37); // ifmOutPWM.PWM1000

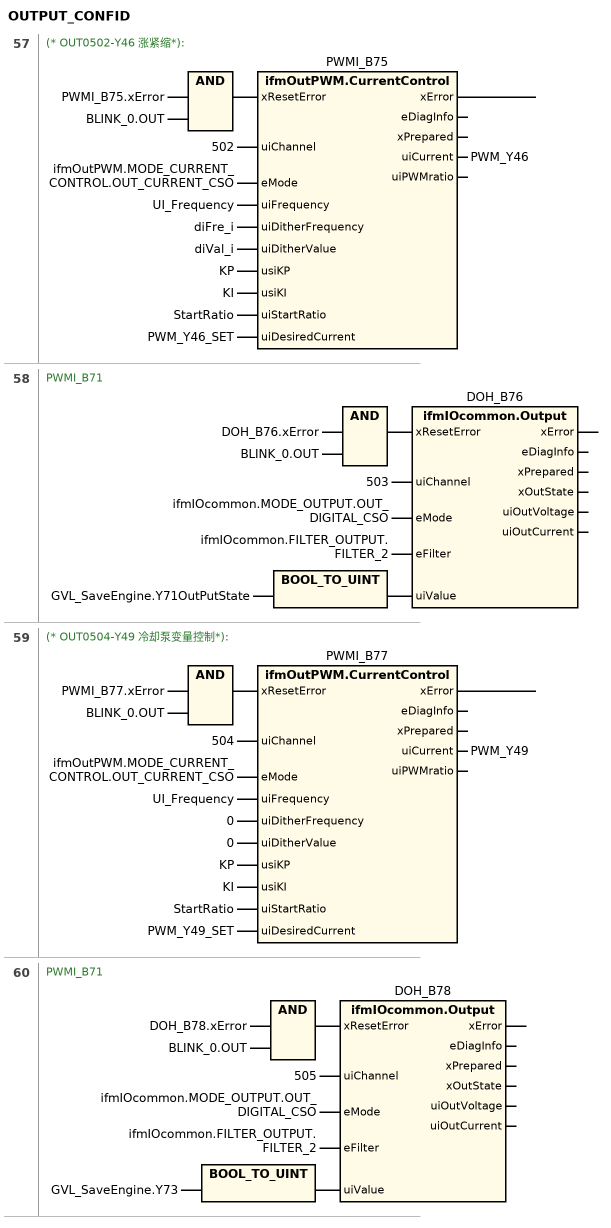
// NETWORK 57
// (* OUT0502-Y46 涨紧缩*):
PWMI_B75(
    xResetError := PWMI_B75.xError AND BLINK_0.OUT,
    uiChannel := 502,
    eMode := ifmOutPWM.MODE_CURRENT_CONTROL.OUT_CURRENT_CSO,
    uiFrequency := UI_Frequency,
    uiDitherFrequency := diFre_i,
    uiDitherValue := diVal_i,
    usiKP := KP,
    usiKI := KI,
    uiStartRatio := StartRatio,
    uiDesiredCurrent := PWM_Y46_SET,
    uiCurrent => PWM_Y46); // ifmOutPWM.CurrentControl

// NETWORK 58
// PWMI_B71
DOH_B76(
    xResetError := DOH_B76.xError AND BLINK_0.OUT,
    uiChannel := 503,
    eMode := ifmIOcommon.MODE_OUTPUT.OUT_DIGITAL_CSO,
    eFilter := ifmIOcommon.FILTER_OUTPUT.FILTER_2,
    uiValue := BOOL_TO_UINT(GVL_SaveEngine.Y71OutPutState)); // ifmIOcommon.Output

// NETWORK 59
// (* OUT0504-Y49 冷却泵变量控制*):
PWMI_B77(
    xResetError := PWMI_B77.xError AND BLINK_0.OUT,
    uiChannel := 504,
    eMode := ifmOutPWM.MODE_CURRENT_CONTROL.OUT_CURRENT_CSO,
    uiFrequency := UI_Frequency,
    uiDitherFrequency := 0,
    uiDitherValue := 0,
    usiKP := KP,
    usiKI := KI,
    uiStartRatio := StartRatio,
    uiDesiredCurrent := PWM_Y49_SET,
    uiCurrent => PWM_Y49); // ifmOutPWM.CurrentControl

// NETWORK 60
// PWMI_B71
DOH_B78(
    xResetError := DOH_B78.xError AND BLINK_0.OUT,
    uiChannel := 505,
    eMode := ifmIOcommon.MODE_OUTPUT.OUT_DIGITAL_CSO,
    eFilter := ifmIOcommon.FILTER_OUTPUT.FILTER_2,
    uiValue := BOOL_TO_UINT(GVL_SaveEngine.Y73)); // ifmIOcommon.Output

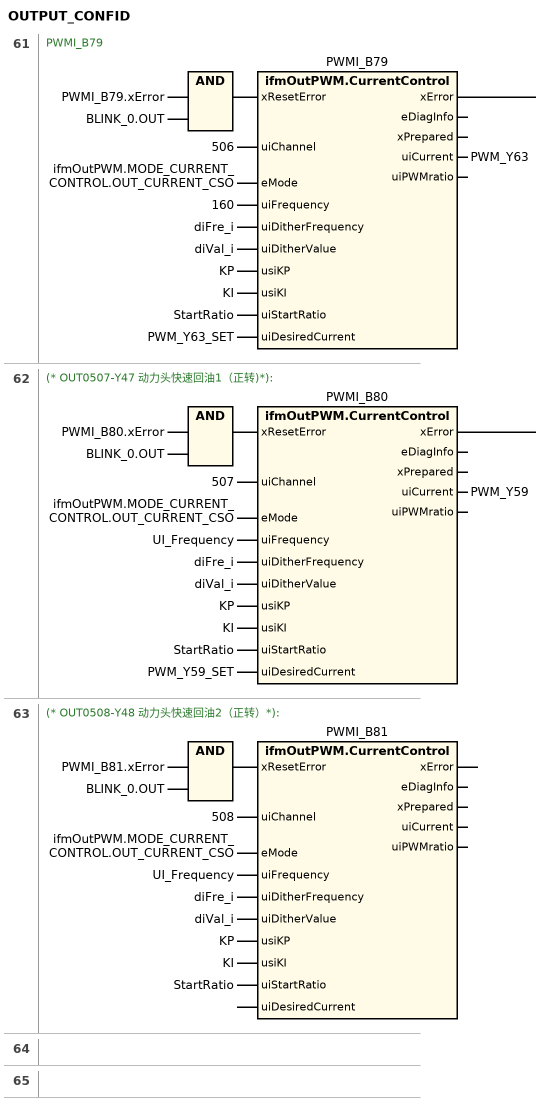
// NETWORK 61
// PWMI_B79
PWMI_B79(
    xResetError := PWMI_B79.xError AND BLINK_0.OUT,
    uiChannel := 506,
    eMode := ifmOutPWM.MODE_CURRENT_CONTROL.OUT_CURRENT_CSO,
    uiFrequency := 160,
    uiDitherFrequency := diFre_i,
    uiDitherValue := diVal_i,
    usiKP := KP,
    usiKI := KI,
    uiStartRatio := StartRatio,
    uiDesiredCurrent := PWM_Y63_SET,
    uiCurrent => PWM_Y63); // ifmOutPWM.CurrentControl

// NETWORK 62
// (* OUT0507-Y47 动力头快速回油1（正转)*):
PWMI_B80(
    xResetError := PWMI_B80.xError AND BLINK_0.OUT,
    uiChannel := 507,
    eMode := ifmOutPWM.MODE_CURRENT_CONTROL.OUT_CURRENT_CSO,
    uiFrequency := UI_Frequency,
    uiDitherFrequency := diFre_i,
    uiDitherValue := diVal_i,
    usiKP := KP,
    usiKI := KI,
    uiStartRatio := StartRatio,
    uiDesiredCurrent := PWM_Y59_SET,
    uiCurrent => PWM_Y59); // ifmOutPWM.CurrentControl

// NETWORK 63
// (* OUT0508-Y48 动力头快速回油2（正转）*):
PWMI_B81(
    xResetError := PWMI_B81.xError AND BLINK_0.OUT,
    uiChannel := 508,
    eMode := ifmOutPWM.MODE_CURRENT_CONTROL.OUT_CURRENT_CSO,
    uiFrequency := UI_Frequency,
    uiDitherFrequency := diFre_i,
    uiDitherValue := diVal_i,
    usiKP := KP,
    usiKI := KI,
    uiStartRatio := StartRatio); // ifmOutPWM.CurrentControl

// NETWORK 64

// NETWORK 65

END_PROGRAM

// StandardPLC/Application/MOVE/Joy_Analog_output
PROGRAM Joy_Analog_output
VAR
	
	Up_Joy_Max:UINT;
	Up_Joy_Min:UINT;
	Down_Joy_Max:UINT;
	Down_Joy_Min:UINT;

	DonglitouAutoMode: BOOL;
END_VAR

Up_Joy_Max:=5000-Par_Joy_DeadBand_max;
Up_Joy_Min:=2500+Par_Joy_DeadBand;
Down_Joy_Min:=Par_Joy_DeadBand_max;
Down_Joy_Max:=2500-Par_Joy_DeadBand;

(*左手柄X方向*)
IF CANI_JOYX_L>Up_Joy_Min AND CANI_JOYX_L<=Up_Joy_Max  THEN
	PWM_JOYX_L_UP:=REAL_TO_UINT((UINT_TO_REAL(CANI_JOYX_L)-2500)/2500*1000);
	PWM_JOYX_L_DOWN:=0;
ELSIF CANI_JOYX_L>Up_Joy_Max THEN(*手柄阶跃*)
	PWM_JOYX_L_UP:=1000;
	PWM_JOYX_L_DOWN:=0;
ELSIF CANI_JOYX_L<=Down_Joy_Max AND CANI_JOYX_L>Down_Joy_Min   THEN
	PWM_JOYX_L_DOWN:=REAL_TO_UINT((2500-UINT_TO_REAL(CANI_JOYX_L))/2500*1000);
	PWM_JOYX_L_UP:=0;
ELSIF CANI_JOYX_L< Down_Joy_Min THEN(*手柄阶跃*)
	PWM_JOYX_L_DOWN:=1000;
	PWM_JOYX_L_UP:=0;
ELSE
	PWM_JOYX_L_UP:=0;
	PWM_JOYX_L_DOWN:=0;
END_IF

(*左手柄Y方向*)
IF CANI_JOYY_L>Up_Joy_Min AND CANI_JOYY_L<=Up_Joy_Max THEN
	PWM_JOYY_L_UP:=REAL_TO_UINT((UINT_TO_REAL(CANI_JOYY_L)-2500)/2500*1000);
	PWM_JOYY_L_DOWN:=0;
ELSIF CANI_JOYY_L>Up_Joy_Max THEN(*手柄阶跃*)
	PWM_JOYY_L_UP:=1000;
	PWM_JOYY_L_DOWN:=0;
ELSIF CANI_JOYY_L<Down_Joy_Max AND CANI_JOYY_L>=Down_Joy_Min THEN
	PWM_JOYY_L_DOWN:=REAL_TO_UINT((2500-UINT_TO_REAL(CANI_JOYY_L))/2500*1000);
	PWM_JOYY_L_UP:=0;
ELSIF CANI_JOYY_L<Down_Joy_Min THEN(*手柄阶跃*)
	PWM_JOYY_L_DOWN:=1000;
	PWM_JOYY_L_UP:=0;
ELSE
	PWM_JOYY_L_UP:=0;
	PWM_JOYY_L_DOWN:=0;
END_IF

(*右手柄X方向*)
IF CANI_JOYX_R>Up_Joy_Min AND CANI_JOYX_R<=Up_Joy_Max THEN
	PWM_JOYX_R_UP:=REAL_TO_UINT((UINT_TO_REAL(CANI_JOYX_R)-2500)/2500*1000);
	PWM_JOYX_R_DOWN:=0;
ELSIF CANI_JOYX_R>Up_Joy_Max THEN(*手柄阶跃*)
	PWM_JOYX_R_UP:=1000;
	PWM_JOYX_R_DOWN:=0;
ELSIF CANI_JOYX_R<Down_Joy_Max AND CANI_JOYX_R>=Down_Joy_Min THEN
	PWM_JOYX_R_DOWN:=REAL_TO_UINT((2500-UINT_TO_REAL(CANI_JOYX_R))/2500*1000);
	PWM_JOYX_R_UP:=0;
ELSIF CANI_JOYX_R<Down_Joy_Min THEN(*手柄阶跃*)
	PWM_JOYX_R_DOWN:=1000;
	PWM_JOYX_R_UP:=0;
ELSE
	PWM_JOYX_R_UP:=0;
	PWM_JOYX_R_DOWN:=0;
END_IF

IF PWM_JOYX_R_DOWN>=100 AND CANI_DongLiTouAutoSwitch AND CANI_WorkModeSwitch THEN
	DonglitouAutoMode:= TRUE;
ELSIF PWM_JOYX_R_UP>=100 OR (NOT CANI_DongLiTouAutoSwitch) OR (NOT CANI_WorkModeSwitch) THEN
	DonglitouAutoMode:= FALSE;
END_IF

IF DonglitouAutoMode THEN
	PWM_JOYX_R_DOWN:=1000;
END_IF
(*右手柄Y方向*)
IF CANI_JOYY_R>Up_Joy_Min AND CANI_JOYY_R<=Up_Joy_Max  THEN
	PWM_JOYY_R_UP:=REAL_TO_UINT((UINT_TO_REAL(CANI_JOYY_R)-2500)/2500*1000);
	PWM_JOYY_R_DOWN:=0;
ELSIF CANI_JOYY_R>Up_Joy_Max THEN(*手柄阶跃*)
	PWM_JOYY_R_UP:=1000;
	PWM_JOYY_R_DOWN:=0;
ELSIF CANI_JOYY_R<Down_Joy_Max  AND CANI_JOYY_R>=Down_Joy_Min THEN
	PWM_JOYY_R_DOWN:=REAL_TO_UINT((2500-UINT_TO_REAL(CANI_JOYY_R))/2500*1000);
	PWM_JOYY_R_UP:=0;
ELSIF CANI_JOYY_R<Down_Joy_Min THEN(*手柄阶跃*)
	PWM_JOYY_R_DOWN:=1000;
	PWM_JOYY_R_UP:=0;
ELSE
	PWM_JOYY_R_UP:=0;
	PWM_JOYY_R_DOWN:=0;
END_IF

(*左脚踏柄*)
IF CANI_JOY_Jiao_L>Up_Joy_Min AND  CANI_JOY_Jiao_L<=Up_Joy_Max  THEN
	PWM_JOY_Jiao_L_UP:=REAL_TO_UINT((UINT_TO_REAL(CANI_JOY_Jiao_L)-2500)/2500*1000);
	PWM_JOY_Jiao_L_DOWN:=0;
ELSIF CANI_JOY_Jiao_L>Up_Joy_Max THEN(*手柄阶跃*)
	PWM_JOY_Jiao_L_UP:=1000;
	PWM_JOY_Jiao_L_DOWN:=0;
ELSIF CANI_JOY_Jiao_L<Down_Joy_Max AND CANI_JOY_Jiao_L>=Down_Joy_Min  THEN
	PWM_JOY_Jiao_L_DOWN:=REAL_TO_UINT((2500-UINT_TO_REAL(CANI_JOY_Jiao_L))/2500*1000);
	PWM_JOY_Jiao_L_UP:=0;
ELSIF CANI_JOY_Jiao_L<Down_Joy_Min THEN(*手柄阶跃*)
	PWM_JOY_Jiao_L_DOWN:=1000;
	PWM_JOY_Jiao_L_UP:=0;
ELSE
	PWM_JOY_Jiao_L_UP:=0;
	PWM_JOY_Jiao_L_DOWN:=0;
END_IF

(*右脚踏柄*)
IF CANI_JOY_Jiao_R>Up_Joy_Min AND CANI_JOY_Jiao_R<=Up_Joy_Max THEN
	PWM_JOY_Jiao_R_UP:=REAL_TO_UINT((UINT_TO_REAL(CANI_JOY_Jiao_R)-2500)/2500*1000);
	PWM_JOY_Jiao_R_DOWN:=0;
ELSIF CANI_JOY_Jiao_R>Up_Joy_Max THEN(*手柄阶跃*)
	PWM_JOY_Jiao_R_UP:=1000;
	PWM_JOY_Jiao_R_DOWN:=0;
ELSIF CANI_JOY_Jiao_R<Down_Joy_Max AND CANI_JOY_Jiao_R>=Down_Joy_Min THEN
	PWM_JOY_Jiao_R_DOWN:=REAL_TO_UINT((2500-UINT_TO_REAL(CANI_JOY_Jiao_R))/2500*1000);
	PWM_JOY_Jiao_R_UP:=0;
ELSIF CANI_JOY_Jiao_R<Down_Joy_Min THEN(*手柄阶跃*)
	PWM_JOY_Jiao_R_DOWN:=1000;
	PWM_JOY_Jiao_R_UP:=0;
ELSE
	PWM_JOY_Jiao_R_UP:=0;
	PWM_JOY_Jiao_R_DOWN:=0;
END_IF

END_PROGRAM

// StandardPLC/Application/CAN/CAN0
PROGRAM CAN0
VAR
	CAN0_INTI: ifmRCAN.CAN_Enable;
	TIME_100ms:TON;
	TIME_200ms:TON;
	TIME_300ms:TON;
	TIME_500ms:TON;
	TIME_700ms:TON;
	TIME_900ms:TON;
	TIME_1000ms:TON;
	TIME_10s:TON;
(*接收*)
(*薄膜按键*)
	CAN1RECEIVE_18F:ifmRCAN.CAN_Rx;
	CAN1RECEIVE_28F:ifmRCAN.CAN_Rx;
	receive_data18F: ARRAY [0..7] OF USINT;
	receive_data28F: ARRAY [0..7] OF USINT;

(*显示屏*)
	CAN1RECEIVE_18E:ifmRCAN.CAN_Rx;
	CAN1RECEIVE_28E:ifmRCAN.CAN_Rx;
	CAN1RECEIVE_38E:ifmRCAN.CAN_Rx;
	CAN1RECEIVE_48E:ifmRCAN.CAN_Rx;
	CAN1RECEIVE_58E:ifmRCAN.CAN_Rx;
	CAN1RECEIVE_68E:ifmRCAN.CAN_Rx;
	CAN1RECEIVE_101:ifmRCAN.CAN_Rx;
	receive_data18E: ARRAY [0..7] OF USINT;
	receive_data28E: ARRAY [0..7] OF USINT;
	receive_data38E: ARRAY [0..7] OF USINT;
	receive_data48E: ARRAY [0..7] OF USINT;
	receive_data58E: ARRAY [0..7] OF USINT;
	receive_data68E: ARRAY [0..7] OF USINT;
	receive_data101: ARRAY [0..7] OF USINT;
	CANI_VAR18E01:UINT;
	CANI_IB_VAR18E0:BYTE;
	CANI_IB_VAR18E1:BOOL;
	CANI_VAR18E23:UINT;
	CANI_VAR18E45:UINT;
	CANI_VAR18E67:UINT;

	CANI_VAR28E01:UINT;
	CANI_IB_VAR28E0:BYTE;
	CANI_IB_VAR28E1:BOOL;
	CANI_VAR28E23:UINT;
	CANI_VAR28E45:UINT;
	CANI_VAR28E67:UINT;

	CANI_VAR38E01:UINT;
	CANI_IB_VAR38E0:BYTE;
	CANI_IB_VAR38E1:BOOL;
	CANI_VAR38E23:UINT;
	CANI_VAR38E45:UINT;
	CANI_VAR38E67:UINT;

	CANI_VAR48E01:UINT;
	CANI_IB_VAR48E0:BYTE;
	CANI_IB_VAR48E1:BOOL;
	CANI_VAR48E23:UINT;
	CANI_VAR48E45:UINT;
	CANI_VAR48E67:UINT;

	CANI_VAR58E01:UINT;
	CANI_IB_VAR58E0:BYTE;
	CANI_IB_VAR58E1:BOOL;
	CANI_VAR58E23:UINT;
	CANI_VAR58E45:UINT;
	CANI_VAR58E67:UINT;

	CANI_VAR68E01:UINT;
	CANI_IB_VAR68E0:BYTE;
	CANI_IB_VAR68E1:BOOL;
	CANI_VAR68E23:UINT;
	CANI_VAR68E45:UINT;
	CANI_VAR68E67:UINT;
(*18E*)
	CANI_IB_VAR00_BOOL: BOOL;
	CANI_IB_VAR01_BOOL: BOOL;
	CANI_IB_VAR02_BOOL: BOOL;
	CANI_IB_VAR03_BOOL: BOOL;
	CANI_IB_VAR04_BOOL: BOOL;
	CANI_IB_VAR05_BOOL: BOOL;
	CANI_IB_VAR06_BOOL: BOOL;
	CANI_IB_VAR07_BOOL: BOOL;
	CANI_IB_VAR08_BOOL: BOOL;
	CANI_IB_VAR09_BOOL: BOOL;
	CANI_IB_VAR10_BOOL: BOOL;
	CANI_IB_VAR11_BOOL: BOOL;
	CANI_IB_VAR12_BOOL: BOOL;
	CANI_IB_VAR13_BOOL: BOOL;
	CANI_IB_VAR14_BOOL: BOOL;
	CANI_IB_VAR15_BOOL: BOOL;
	CANI_IB_VAR30_BOOL:BOOL;
	CANI_IB_VAR33_BOOL:BOOL;
	CANI_IB_VAR33_BOOL_2:BOOL;
	CANI_IB_VAR33_BOOL_3:BOOL;
	CANI_IB_VAR33_BOOL_4:BOOL;
	CANI_IB_VAR34_BOOL:BOOL;
	CANI_IB_VAR36_BOOL:BOOL;
	CANI_IB_VAR37_BOOL:BOOL;
	CANI_IB_VAR38_BOOL:BOOL;
	CANI_IB_VAR40_BOOL:BOOL;
	CANI_IB_VAR41_BOOL:BOOL;
	CANI_IB_VAR42_BOOL:BOOL;
	CANI_IB_VAR42_BOOL_2:BOOL;
	CANI_IB_VAR42_BOOL_3:BOOL;
	CANI_IB_VAR42_BOOL_4:BOOL;
	CANI_IB_VAR42_BOOL_5:BOOL;
	CANI_IB_VAR43_BOOL:BOOL;
	CANI_IB_VAR43_BOOL_2:BOOL;
	CANI_IB_VAR48_BOOL:BOOL;
	CANI_IB_VAR80_BOOL: BOOL;//节能0x50,
	
	CANI_IB_VAR9_BOOL_2:BOOL;
	CANI_IB_VAR9_BOOL_3:BOOL;
	CANI_IB_VAR9_BOOL_4:BOOL;
	
	CANI_IB_VAR11_BOOL_2: BOOL;
	CANI_IB_VAR11_BOOL_3: BOOL;
	CANI_IB_VAR11_BOOL_4: BOOL;
	CANI_IB_VAR11_BOOL_5: BOOL;

	CANI_IB_VAR16_BOOL: BOOL;
	CANI_IB_VAR16_BOOL_2: BOOL;
	CANI_IB_VAR16_BOOL_3: BOOL;
	CANI_IB_VAR16_BOOL_4: BOOL;
	
	CANI_IB_VAR17_BOOL: BOOL;	
	
	CANI_IB_VAR8_BOOL_2: BOOL;
	CANI_IB_VAR8_BOOL_3: BOOL;
	CANI_IB_VAR8_BOOL_4: BOOL;
	
//发送	
	send_data187:ARRAY [0..7] OF USINT;
	send_data287:ARRAY [0..7] OF USINT;
	send_data387:ARRAY [0..7] OF USINT;
	send_data487:ARRAY [0..7] OF USINT;
	send_data587:ARRAY [0..7] OF USINT;
	send_data687:ARRAY [0..7] OF USINT;
	send_data787:ARRAY [0..7] OF USINT;
	send_data188:ARRAY [0..7] OF USINT;
	send_data288:ARRAY [0..7] OF USINT;
	send_data388:ARRAY [0..7] OF USINT;
	send_data488:ARRAY [0..7] OF USINT;
	send_data189:ARRAY [0..7] OF USINT;
	send_data289:ARRAY [0..7] OF USINT;
	send_data389:ARRAY [0..7] OF USINT;
	send_data489:ARRAY [0..7] OF USINT;
	send_data18A:ARRAY [0..7] OF USINT;
	send_data28A:ARRAY [0..7] OF USINT;
	send_data38A:ARRAY [0..7] OF USINT;
	send_data48A:ARRAY [0..7] OF USINT;
	send_data18B:ARRAY [0..7] OF USINT;
	send_data28B:ARRAY [0..7] OF USINT;
	send_data38B:ARRAY [0..7] OF USINT;
	send_data48B:ARRAY [0..7] OF USINT;
	send_data18C:ARRAY [0..7] OF USINT;
	send_data28C:ARRAY [0..7] OF USINT;
	send_data38C:ARRAY [0..7] OF USINT;
	send_data48C:ARRAY [0..7] OF USINT;
	send_data18D:ARRAY [0..7] OF USINT;
	send_data28D:ARRAY [0..7] OF USINT;
	send_data38D:ARRAY [0..7] OF USINT;
	send_data48D:ARRAY [0..7] OF USINT;
	send_data186:ARRAY [0..7] OF USINT;
	send_data286:ARRAY [0..7] OF USINT;
	send_data386:ARRAY [0..7] OF USINT;
	send_data486:ARRAY [0..7] OF USINT;
	send_data586:ARRAY [0..7] OF USINT;
	send_data686:ARRAY [0..7] OF USINT;
	send_data786:ARRAY [0..7] OF USINT;
	send_data185:ARRAY [0..7] OF USINT;
	send_data285:ARRAY [0..7] OF USINT;
	send_data385:ARRAY [0..7] OF USINT;
	send_data485:ARRAY [0..7] OF USINT;
	send_data585:ARRAY [0..7] OF USINT;
	send_data685:ARRAY [0..7] OF USINT;
	send_data785:ARRAY [0..7] OF USINT;
	send_data184:ARRAY [0..7] OF USINT;
	send_data284:ARRAY [0..7] OF USINT;
	send_data384:ARRAY [0..7] OF USINT;
	send_data484:ARRAY [0..7] OF USINT;
	send_data584:ARRAY [0..7] OF USINT;
	send_data684:ARRAY [0..7] OF USINT;
	send_data784:ARRAY [0..7] OF USINT;
	send_data381:ARRAY [0..7] OF USINT;
	send_data481:ARRAY [0..7] OF USINT;
	send_data581:ARRAY [0..7] OF USINT;
	send_data681:ARRAY [0..7] OF USINT;
	send_data781:ARRAY [0..7] OF USINT;
	send_data182:ARRAY [0..7] OF USINT;
	send_data183:ARRAY [0..7] OF USINT;
	send_data283:ARRAY [0..7] OF USINT;
	send_data102:ARRAY [0..7] OF USINT;
	
	//节能
	send_data18F00001:ARRAY [0..7] OF USINT;
	send_data18F00002:ARRAY [0..7] OF USINT;
	
	CAN1_SEND_187:ifmRCAN.CAN_Tx;
	CAN1_SEND_287:ifmRCAN.CAN_Tx;
	CAN1_SEND_387:ifmRCAN.CAN_Tx;
	CAN1_SEND_487:ifmRCAN.CAN_Tx;
	CAN1_SEND_587:ifmRCAN.CAN_Tx;
	CAN1_SEND_687:ifmRCAN.CAN_Tx;
	CAN1_SEND_787:ifmRCAN.CAN_Tx;
	CAN1_SEND_188:ifmRCAN.CAN_Tx;
	CAN1_SEND_288:ifmRCAN.CAN_Tx;
	CAN1_SEND_388:ifmRCAN.CAN_Tx;
	CAN1_SEND_488:ifmRCAN.CAN_Tx;
	CAN1_SEND_189:ifmRCAN.CAN_Tx;
	CAN1_SEND_289:ifmRCAN.CAN_Tx;
	CAN1_SEND_389:ifmRCAN.CAN_Tx;
	CAN1_SEND_489:ifmRCAN.CAN_Tx;
	CAN1_SEND_18A:ifmRCAN.CAN_Tx;
	CAN1_SEND_28A:ifmRCAN.CAN_Tx;
	CAN1_SEND_38A:ifmRCAN.CAN_Tx;
	CAN1_SEND_48A:ifmRCAN.CAN_Tx;
	CAN1_SEND_18B:ifmRCAN.CAN_Tx;
	CAN1_SEND_28B:ifmRCAN.CAN_Tx;
	CAN1_SEND_38B:ifmRCAN.CAN_Tx;
	CAN1_SEND_48B:ifmRCAN.CAN_Tx;
	CAN1_SEND_18C:ifmRCAN.CAN_Tx;
	CAN1_SEND_28C:ifmRCAN.CAN_Tx;
	CAN1_SEND_38C:ifmRCAN.CAN_Tx;
	CAN1_SEND_48C:ifmRCAN.CAN_Tx;
	CAN1_SEND_18D:ifmRCAN.CAN_Tx;
	CAN1_SEND_28D:ifmRCAN.CAN_Tx;
	CAN1_SEND_38D:ifmRCAN.CAN_Tx;
	CAN1_SEND_48D:ifmRCAN.CAN_Tx;
	CAN1_SEND_186:ifmRCAN.CAN_Tx;
	CAN1_SEND_286:ifmRCAN.CAN_Tx;
	CAN1_SEND_386:ifmRCAN.CAN_Tx;
	CAN1_SEND_486:ifmRCAN.CAN_Tx;
	CAN1_SEND_586:ifmRCAN.CAN_Tx;
	CAN1_SEND_686:ifmRCAN.CAN_Tx;
	CAN1_SEND_786:ifmRCAN.CAN_Tx;
	CAN1_SEND_185:ifmRCAN.CAN_Tx;
	CAN1_SEND_285:ifmRCAN.CAN_Tx;
	CAN1_SEND_385:ifmRCAN.CAN_Tx;
	CAN1_SEND_485:ifmRCAN.CAN_Tx;
	CAN1_SEND_585:ifmRCAN.CAN_Tx;
	CAN1_SEND_685:ifmRCAN.CAN_Tx;
	CAN1_SEND_785:ifmRCAN.CAN_Tx;
	CAN1_SEND_184:ifmRCAN.CAN_Tx;
	CAN1_SEND_284:ifmRCAN.CAN_Tx;
	CAN1_SEND_384:ifmRCAN.CAN_Tx;
	CAN1_SEND_484:ifmRCAN.CAN_Tx;
	CAN1_SEND_584:ifmRCAN.CAN_Tx;
	CAN1_SEND_684:ifmRCAN.CAN_Tx;
	CAN1_SEND_784:ifmRCAN.CAN_Tx;
	CAN1_SEND_381:ifmRCAN.CAN_Tx;
	CAN1_SEND_481:ifmRCAN.CAN_Tx;
	CAN1_SEND_581:ifmRCAN.CAN_Tx;
	CAN1_SEND_681:ifmRCAN.CAN_Tx;
	CAN1_SEND_781:ifmRCAN.CAN_Tx;
	CAN1_SEND_182:ifmRCAN.CAN_Tx;
	CAN1_SEND_183:ifmRCAN.CAN_Tx;
	CAN1_SEND_283:ifmRCAN.CAN_Tx;
	CAN1_SEND_102:ifmRCAN.CAN_Tx;
	//节能
	CAN1_SEND_18F00001:ifmRCAN.CAN_Tx;
	CAN1_SEND_18F00002:ifmRCAN.CAN_Tx;
	
	x1:DINT;
	x2:DINT;
	d1:DINT;
	d2:DINT;
	tCounter:UINT;
	temp_bool1:BOOL;
	tp_20s:tp;
END_VAR

(*CAN1口使能及初始化*)	
CAN0_INTI(xEnable:=NOT init_1 , eChannel:=ifmRCAN.ifmDevice.CHAN_0, eBaudrate:=ifmRCAN.ifmDevice.CAN_BAUDRATE.KBAUD_250 );	
//CANbus_0();
(*CAN1口 接显示屏 薄膜按键 *)
(***********接收************)
(*薄膜按键*)
CAN1RECEIVE_18F(xEnable:=TRUE , eChannel:= 0, xExtended:= FALSE, aData=> receive_data18F, udiID:= 16#18F);
(*BYTE0*)
CANI_WorkModeSwitch:=BYTE_TO_BOOL(receive_data18F[0] AND 2#00000001);
CANI_MaiWinFloatSwitch:=BYTE_TO_BOOL(receive_data18F[0] AND 2#00000010);
CANI_ColdFunSwitch:=BYTE_TO_BOOL(receive_data18F[0] AND 2#00000100);
CANI_DonglitouLSwitch:=BYTE_TO_BOOL(receive_data18F[0] AND 2#00001000);
CANI_DonglitouMSwitch:=BYTE_TO_BOOL(receive_data18F[0] AND 2#00010000);
CANI_DonglitouHSwitch:=BYTE_TO_BOOL(receive_data18F[0] AND 2#00100000);
CANI_IdleEnbleSwitch:=BYTE_TO_BOOL(receive_data18F[0] AND 2#01000000);
CANI_DongLiTouPressLimitSwitch:=BYTE_TO_BOOL(receive_data18F[0] AND 2#10000000);
(*BYTE1*)
CANI_DonglitouADDSwitch:=BYTE_TO_BOOL(receive_data18F[1] AND 2#00000001);
CANI_DonglitouSUBSwitch:=BYTE_TO_BOOL(receive_data18F[1] AND 2#00000010);
CANI_MoShiSwitch:=BYTE_TO_BOOL(receive_data18F[1] AND 2#00000100);
CANI_CFASwitch:=BYTE_TO_BOOL(receive_data18F[1] AND 2#00001000);
CANI_RotationSuoSwitch:=BYTE_TO_BOOL(receive_data18F[1] AND 2#00010000);
CANI_RotationShenSwitch:=BYTE_TO_BOOL(receive_data18F[1] AND 2#00100000);
CANI_ShengZhangJinSwitch:=BYTE_TO_BOOL(receive_data18F[1] AND 2#01000000);
CANI_LvDaiShenSuoSwitch:=BYTE_TO_BOOL(receive_data18F[1] AND 2#10000000);
(*BYTE2*)
CANI_ETouYouGangSwitch:=BYTE_TO_BOOL(receive_data18F[2] AND 2#00000001);
CANI_MidSpeedSwitch:=BYTE_TO_BOOL(receive_data18F[2] AND 2#00000010);
CANI_ECOSwitch:=BYTE_TO_BOOL(receive_data18F[2] AND 2#00000100);
CANI_DongLiTouSpeedSlowSwitch:=BYTE_TO_BOOL(receive_data18F[2] AND 2#01000000);
//CANI_JiaYaFastSwitch:=BYTE_TO_BOOL(receive_data18F[2] AND 2#10000000);
CANI_DongLiTouAutoSwitch:=BYTE_TO_BOOL(receive_data18F[2] AND 2#00001000);


(*显示屏值*)
CAN1RECEIVE_18E(xEnable:=TRUE , eChannel:= 0, xExtended:= FALSE, aData=> receive_data18E, udiID:= 16#18E);
CANI_IB_VAR18E0:=receive_data18E[0];
CANI_IB_VAR18E1:=BYTE_TO_BOOL(receive_data18E[1] AND 2#00000001);
CANI_VAR18E01:=receive_data18E[0]+receive_data18E[1]*256;
CANI_VAR18E23:=receive_data18E[2]+receive_data18E[3]*256;
CANI_VAR18E45:=receive_data18E[4]+receive_data18E[5]*256;
CANI_VAR18E67:=receive_data18E[6]+receive_data18E[7]*256;

CAN1RECEIVE_28E(xEnable:=TRUE , eChannel:= 0, xExtended:= FALSE, aData=> receive_data28E, udiID:= 16#28E);
CANI_IB_VAR28E0:=receive_data28E[0];
CANI_IB_VAR28E1:=BYTE_TO_BOOL(receive_data28E[1] AND 2#00000001);
CANI_VAR28E01:=receive_data28E[0]+receive_data28E[1]*256;
CANI_VAR28E23:=receive_data28E[2]+receive_data28E[3]*256;
CANI_VAR28E45:=receive_data28E[4]+receive_data28E[5]*256;
CANI_VAR28E67:=receive_data28E[6]+receive_data28E[7]*256;

CAN1RECEIVE_38E(xEnable:=TRUE , eChannel:= 0, xExtended:= FALSE, aData=> receive_data38E, udiID:= 16#38E);
CANI_IB_VAR38E0:=receive_data38E[0];
CANI_IB_VAR38E1:=BYTE_TO_BOOL(receive_data38E[1] AND 2#00000001);
CANI_VAR38E01:=receive_data38E[0]+receive_data38E[1]*256;
CANI_VAR38E23:=receive_data38E[2]+receive_data38E[3]*256;
CANI_VAR38E45:=receive_data38E[4]+receive_data38E[5]*256;
CANI_VAR38E67:=receive_data38E[6]+receive_data38E[7]*256;

CAN1RECEIVE_48E(xEnable:=TRUE , eChannel:= 0, xExtended:= FALSE, aData=> receive_data48E, udiID:= 16#48E);
CANI_IB_VAR48E0:=receive_data48E[0];
CANI_IB_VAR48E1:=BYTE_TO_BOOL(receive_data48E[1] AND 2#00000001);
CANI_VAR48E01:=receive_data48E[0]+receive_data48E[1]*256;
CANI_VAR48E23:=receive_data48E[2]+receive_data48E[3]*256;
CANI_VAR48E45:=receive_data48E[4]+receive_data48E[5]*256;
CANI_VAR48E67:=receive_data48E[6]+receive_data48E[7]*256;

CAN1RECEIVE_58E(xEnable:=TRUE , eChannel:= 0, xExtended:= FALSE, aData=> receive_data58E, udiID:= 16#58E);
CANI_IB_VAR58E0:=receive_data58E[0];
CANI_IB_VAR58E1:=BYTE_TO_BOOL(receive_data58E[1] AND 2#00000001);
CANI_VAR58E01:=receive_data58E[0]+receive_data58E[1]*256;
CANI_VAR58E23:=receive_data58E[2]+receive_data58E[3]*256;
CANI_VAR58E45:=receive_data58E[4]+receive_data58E[5]*256;
CANI_VAR58E67:=receive_data58E[6]+receive_data58E[7]*256;

CAN1RECEIVE_68E(xEnable:=TRUE , eChannel:= 0, xExtended:= FALSE, aData=> receive_data68E, udiID:= 16#68E);
CANI_IB_VAR68E0:=receive_data68E[0];
CANI_IB_VAR68E1:=BYTE_TO_BOOL(receive_data68E[1] AND 2#00000001);
CANI_VAR68E01:=receive_data68E[0]+receive_data68E[1]*256;
CANI_VAR68E23:=receive_data68E[2]+receive_data68E[3]*256;
CANI_VAR68E45:=receive_data68E[4]+receive_data68E[5]*256;
CANI_VAR68E67:=receive_data68E[6]+receive_data68E[7]*256;




(*施工桩号及直径*)
PileDiameter:=CANI_VAR68E23;
PileNumble:=CANI_VAR68E45;
(*18E标志位*)
CANI_IB_VAR00_BOOL:=CANI_IB_VAR18E0=0;
CANI_IB_VAR01_BOOL:=CANI_IB_VAR18E0=1;
CANI_IB_VAR02_BOOL:=CANI_IB_VAR18E0=2;
CANI_IB_VAR03_BOOL:=CANI_IB_VAR18E0=3;
CANI_IB_VAR05_BOOL:=CANI_IB_VAR18E0=5;
CANI_IB_VAR06_BOOL:=CANI_IB_VAR18E0=6;
CANI_IB_VAR07_BOOL:=CANI_IB_VAR18E0=7;
CANI_IB_VAR08_BOOL:=CANI_IB_VAR18E0=8;
CANI_IB_VAR09_BOOL:=CANI_IB_VAR18E0=9;
CANI_IB_VAR10_BOOL:=CANI_IB_VAR18E0=10;
CANI_IB_VAR11_BOOL:=CANI_IB_VAR18E0=11;
CANI_IB_VAR12_BOOL:=CANI_IB_VAR18E0=12;
CANI_IB_VAR13_BOOL:=CANI_IB_VAR18E0=13;
CANI_IB_VAR14_BOOL:=CANI_IB_VAR18E0=14;
CANI_IB_VAR15_BOOL:=CANI_IB_VAR18E0=15;
CANI_IB_VAR16_BOOL:=CANI_IB_VAR18E0=16;
CANI_IB_VAR17_BOOL:=CANI_IB_VAR18E0=17;
CANI_IB_VAR30_BOOL:=CANI_IB_VAR18E0=30;
CANI_IB_VAR33_BOOL:=CANI_IB_VAR18E0=33;
CANI_IB_VAR34_BOOL:=CANI_IB_VAR18E0=34;
CANI_IB_VAR36_BOOL:=CANI_IB_VAR18E0=36;
CANI_IB_VAR37_BOOL:=CANI_IB_VAR18E0=37;
CANI_IB_VAR38_BOOL:=CANI_IB_VAR18E0=38;
CANI_IB_VAR40_BOOL:=CANI_IB_VAR18E0=40;
CANI_IB_VAR41_BOOL:=CANI_IB_VAR18E0=41;
CANI_IB_VAR42_BOOL:=CANI_IB_VAR18E0=42;
CANI_IB_VAR43_BOOL:=CANI_IB_VAR18E0=43;
CANI_IB_VAR48_BOOL:=CANI_IB_VAR18E0=48;
//节能0x50=80,2字节节能开关，3字节泄压开关
CANI_IB_VAR80_BOOL:=CANI_IB_VAR18E0=80;
(*28E标志位*)
CANI_IB_VAR8_BOOL_2:=CANI_IB_VAR28E0=8;
CANI_IB_VAR9_BOOL_2:=CANI_IB_VAR28E0=9;
CANI_IB_VAR11_BOOL_2:=CANI_IB_VAR28E0=11;
CANI_IB_VAR16_BOOL_2:=CANI_IB_VAR28E0=16;
CANI_IB_VAR33_BOOL_2:=CANI_IB_VAR28E0=33;
CANI_IB_VAR42_BOOL_2:=CANI_IB_VAR28E0=42;
CANI_IB_VAR43_BOOL_2:=CANI_IB_VAR28E0=43;
(*38E标志位*)
CANI_IB_VAR8_BOOL_3:=CANI_IB_VAR38E0=8;
CANI_IB_VAR9_BOOL_3:=CANI_IB_VAR38E0=9;
CANI_IB_VAR11_BOOL_3:=CANI_IB_VAR38E0=11;
CANI_IB_VAR16_BOOL_3:=CANI_IB_VAR38E0=16;
CANI_IB_VAR33_BOOL_3:=CANI_IB_VAR38E0=33;
CANI_IB_VAR42_BOOL_3:=CANI_IB_VAR38E0=42;
(*48E标志位*)
CANI_IB_VAR8_BOOL_4:=CANI_IB_VAR48E0=8;
CANI_IB_VAR9_BOOL_4:=CANI_IB_VAR48E0=9;
CANI_IB_VAR11_BOOL_4:=CANI_IB_VAR48E0=11;
CANI_IB_VAR16_BOOL_4:=CANI_IB_VAR48E0=16;
CANI_IB_VAR33_BOOL_4:=CANI_IB_VAR48E0=33;
(*58E标志位*)
CANI_IB_VAR11_BOOL_5:=CANI_IB_VAR58E0=11;

(*PID设置界面*)
IF CANI_IB_VAR00_BOOL AND CANI_IB_VAR18E1 THEN
	IF CANI_VAR18E45<>0 THEN
		PAR_KP:=CANI_VAR18E45;
	END_IF
	IF CANI_VAR18E67<>0 THEN
		PAR_KI:=UINT_TO_BYTE(CANI_VAR18E67);
	END_IF
END_IF
IF CANI_IB_VAR01_BOOL AND CANI_IB_VAR18E1 THEN
	IF CANI_VAR18E23<>0 THEN
		PAR_KD:=UINT_TO_BYTE(CANI_VAR18E23);
	END_IF
	IF CANI_VAR18E45<>0 THEN
		PAR_Y27_PosFull:=CANI_VAR18E45;(*阀A正向最大*)
	END_IF
	IF CANI_VAR18E67<>0 THEN
		PAR_Y27_NegFull:=CANI_VAR18E67;(*阀A正向最小*)
	END_IF
END_IF
IF CANI_IB_VAR02_BOOL AND CANI_IB_VAR18E1 THEN
	IF CANI_VAR18E23<>0 THEN
		PAR_Y28_PosFull:=CANI_VAR18E23;(*阀A逆向最大*)
	END_IF
	IF CANI_VAR18E45<>0 THEN
		PAR_Y28_NegFull:=CANI_VAR18E45;(*阀A逆向最小*)
	END_IF
	IF CANI_VAR18E67<>0 THEN
		PAR_Y29_PosFull:=CANI_VAR18E67;(*阀B正向最大*)
	END_IF
END_IF
IF CANI_IB_VAR03_BOOL AND CANI_IB_VAR18E1 THEN
	IF CANI_VAR18E23<>0 THEN
		PAR_Y29_NegFull:=CANI_VAR18E23;(*阀B正向最小*)
	END_IF
	IF CANI_VAR18E45<>0 THEN
		PAR_Y30_PosFull:=CANI_VAR18E45;(*阀B逆向最大*)
	END_IF
	IF CANI_VAR18E67<>0 THEN
		PAR_Y30_NegFull:=CANI_VAR18E67;(*阀B逆向最小*)
	END_IF
END_IF

(*调平界面*)
IF CANI_IB_VAR05_BOOL AND CANI_IB_VAR18E1 THEN
	CANI_Button_LEVER_Auto:=BYTE_TO_BOOL(receive_data18E[2] AND 2#00000001);
	CANI_Button_LEVER_XPlus:=BYTE_TO_BOOL(receive_data18E[3] AND 2#00000001);
	CANI_Button_LEVER_XSubtract:=BYTE_TO_BOOL(receive_data18E[4] AND 2#00000001);
	CANI_Button_LEVER_YPlus:=BYTE_TO_BOOL(receive_data18E[5] AND 2#00000001);
	CANI_Button_LEVER_YSubtract:=BYTE_TO_BOOL(receive_data18E[6] AND 2#00000001);
	CANI_Button_LEVER_Manual:=BYTE_TO_BOOL(receive_data18E[7] AND 2#00000001);
END_IF

(*主界面*)
IF CANI_IB_VAR06_BOOL AND CANI_IB_VAR18E1 THEN
	CANI_Button_RotationOriginal:=BYTE_TO_BOOL(receive_data18E[2] AND 2#00000001);
	CANI_Button_DepthClear:=BYTE_TO_BOOL(receive_data18E[3] AND 2#00000001);
	CANI_Button_BuzzSwitch:=BYTE_TO_BOOL(receive_data18E[4] AND 2#00000001);
	CANI_Button_FloatSwitch:=BYTE_TO_BOOL(receive_data18E[5] AND 2#00000001);
END_IF

(*调试界面*)
IF CANI_IB_VAR07_BOOL AND CANI_IB_VAR18E1 THEN
	CANI_Button_Debug_LStretchOut:=BYTE_TO_BOOL(receive_data18E[2] AND 2#00000001);
	CANI_Button_Debug_LRetraction:=BYTE_TO_BOOL(receive_data18E[3] AND 2#00000001);
	CANI_Button_Debug_RStretchOut:=BYTE_TO_BOOL(receive_data18E[4] AND 2#00000001);
	CANI_Button_Debug_RRetraction:=BYTE_TO_BOOL(receive_data18E[5] AND 2#00000001);
END_IF

(*参数设置界面*)
(*IF CANI_IB_VAR08_BOOL AND CANI_IB_VAR18E1 THEN
	IF CANI_VAR18E23<>0 THEN
		PAR_MainAngleSetting:=CANI_VAR18E23;
	END_IF
	IF CANI_VAR18E67<>0 THEN
		PAR_RotationPercision:=CANI_VAR18E67;
	END_IF
END_IF*)

IF CANI_IB_VAR8_BOOL_2 AND CANI_IB_VAR28E1 THEN
	IF CANI_VAR28E23<>0 THEN
		PAR_Speed_Idling:=CANI_VAR18E23;
	END_IF
END_IF

IF CANI_IB_VAR8_BOOL_3 AND CANI_IB_VAR38E1 THEN
	CANI_Button_Zero_AngleX:=BYTE_TO_BOOL(receive_data38E[2] AND 2#00000001);
	CANI_Button_Zero_AngleY:=BYTE_TO_BOOL(receive_data38E[3] AND 2#00000001);
END_IF

IF CANI_IB_VAR8_BOOL_4 AND CANI_IB_VAR48E1 THEN
	PAR_Circle1:=CANI_VAR48E23;
	IF CANI_VAR48E45<>0 THEN
		PAR_Circle2:=CANI_VAR48E45;
	END_IF
	IF CANI_VAR48E67<>0 THEN
		PAR_Quanshu:=CANI_VAR48E67;
	END_IF
END_IF

(*手柄设置*)
IF CANI_IB_VAR09_BOOL AND CANI_IB_VAR18E1 THEN
	IF CANI_VAR18E45<>0 THEN
		PAR_M_Joy_LEN:=CANI_VAR18E45;
	END_IF
	IF CANI_VAR18E67<>0 THEN
		PAR_DeadBand_x:=CANI_VAR18E67;
	END_IF
END_IF
IF CANI_IB_VAR9_BOOL_2 AND CANI_IB_VAR28E1 THEN
	IF CANI_VAR28E23<>0 THEN
		PAR_PosFull_x:=CANI_VAR28E23;
	END_IF
	IF CANI_VAR28E45<>0 THEN
		PAR_NegFull_x:=CANI_VAR28E45;
	END_IF
	IF CANI_VAR28E67<>0 THEN
		PAR_Progression_x:=CANI_VAR28E67;
	END_IF
END_IF
IF CANI_IB_VAR9_BOOL_3 AND CANI_IB_VAR38E1 THEN
	IF CANI_VAR38E23<>0 THEN
		PAR_DeadBand_y:=CANI_VAR38E23;
	END_IF
	IF CANI_VAR38E45<>0 THEN
		PAR_PosFull_y:=CANI_VAR38E45;
	END_IF
	IF CANI_VAR38E67<>0 THEN
		PAR_NegFull_y:=CANI_VAR38E67;
	END_IF
END_IF
IF CANI_IB_VAR9_BOOL_4 AND CANI_IB_VAR48E1 THEN
	IF CANI_VAR48E23<>0 THEN
		PAR_Progression_y:=CANI_VAR48E23;
	END_IF
	IF CANI_VAR48E45<>0 THEN
		PAR_Zero_x:=CANI_VAR48E45;
	END_IF
	IF CANI_VAR48E67<>0 THEN
		PAR_Zero_y:=CANI_VAR48E67;
	END_IF
END_IF

(*步长设置界面*)
IF CANI_IB_VAR10_BOOL AND CANI_IB_VAR18E1 THEN
	IF CANI_VAR18E23<>0 THEN
		PAR_ControlValue:=CANI_VAR18E23;
	END_IF
END_IF
(*报警设置界面*)
IF NOT CANI_IB_VAR11_BOOL THEN
	CANI_IB_VAR11_BOOL_2:= FALSE;
	CANI_IB_VAR11_BOOL_3:= FALSE;
	CANI_IB_VAR11_BOOL_4:= FALSE;
	CANI_IB_VAR11_BOOL_5:= FALSE;
END_IF

IF CANI_IB_VAR11_BOOL AND CANI_IB_VAR18E1 THEN
	IF CANI_VAR18E23<>0 THEN
		PAR_WarnFuelLevel_Low:=CANI_VAR18E23;(*燃油液位低报警值*)
	END_IF
	IF CANI_VAR18E45<>0 THEN
		PAR_WarnHydOilTem_High:=CANI_VAR18E45;(*液压油温高报警值*)
	END_IF
END_IF

IF CANI_IB_VAR11_BOOL_2 AND CANI_IB_VAR28E1 THEN
	IF CANI_VAR28E23<>0 THEN
		PAR_WarnOilPress_Low:=CANI_VAR28E23;(*机油压力低报警值*)
	END_IF
	IF CANI_VAR28E67<>0 THEN
		PAR_WarnWaterTem_High:=CANI_VAR28E67;(*冷却水温高报警值*)
	END_IF
END_IF

IF CANI_IB_VAR11_BOOL_3 AND CANI_IB_VAR38E1 THEN
	IF CANI_VAR38E45<>0 THEN
		PAR_HydOilPress_PosFull:=CANI_VAR38E45;(*压力传感器上限值*)
	END_IF
	IF CANI_VAR38E67<>0 THEN
		PAR_HydOilPress_NegFull:=CANI_VAR38E67;(*压力传感器下限值*)
	END_IF
END_IF

IF CANI_IB_VAR11_BOOL_4 AND CANI_IB_VAR48E1 THEN
	IF CANI_VAR48E23<>0 THEN
		PAR_HydOilPilotPress_PosFull:=CANI_VAR48E23;(*先导压力传感器上限值*)
	END_IF
	IF CANI_VAR48E45<>0 THEN
		PAR_HydOilPilotPress_NegFull:=CANI_VAR48E45;(*先导压力传感器下限值*)
	END_IF
	IF CANI_VAR48E67<>0 THEN
		PAR_WarnTension_High:=CANI_VAR48E67;(*拉力超限设置值*)
	END_IF
END_IF

IF CANI_IB_VAR11_BOOL_5 AND CANI_IB_VAR58E1 THEN
	IF CANI_VAR58E23<>0 THEN
		PAR_TensionSensor_PosFull:=CANI_VAR58E23;(*拉力传感器上限值*)
	END_IF
	IF CANI_VAR58E45<>0 THEN
		PAR_TensionSensor_NegFull:=CANI_VAR58E45;(*拉力传感器下限值*)
	END_IF
	IF CANI_VAR58E67<>0 THEN
		PAR_TensionSensor_Range:=CANI_VAR58E67;(*拉力传感器量程*)
	END_IF
END_IF
(*记录清零界面*)
IF CANI_IB_VAR14_BOOL AND CANI_IB_VAR18E1 THEN
	CANI_Button_RecordClear1:=BYTE_TO_BOOL(receive_data18E[2] AND 2#00000001);
	//CANI_Button_RecordClear:=BYTE_TO_BOOL(receive_data18E[2] AND 2#00000001);
END_IF
(*回转设置界面*)
IF CANI_IB_VAR16_BOOL AND CANI_IB_VAR18E1 THEN
	IF CANI_VAR18E23<>0 THEN
		PAR_Sudu1_Min:=CANI_VAR18E23;
	END_IF
	IF CANI_VAR18E45<>0 THEN
		PAR_Sudu1_Max:=CANI_VAR18E45;
	END_IF
	IF CANI_VAR18E67<>0 THEN
		PAR_Sudu1_Middle:=CANI_VAR18E67;
	END_IF
END_IF
IF CANI_IB_VAR16_BOOL_2 AND CANI_IB_VAR28E1 THEN
	IF CANI_VAR28E23<>0 THEN
		PAR_Angle1:=CANI_VAR28E23;
	END_IF
	IF CANI_VAR28E45<>0 THEN
		PAR_Angle2:=CANI_VAR28E45;
	END_IF
	IF CANI_VAR28E67<>0 THEN
		PAR_Angle3:=CANI_VAR28E67;
	END_IF
END_IF

IF CANI_IB_VAR16_BOOL_3 AND CANI_IB_VAR38E1 THEN
	IF CANI_VAR38E23<>0 THEN
		PAR_Sudu2_Min:=CANI_VAR38E23;
	END_IF
	IF CANI_VAR38E45<>0 THEN
		PAR_Sudu2_Max:=CANI_VAR38E45;
	END_IF
	IF CANI_VAR38E67<>0 THEN
		PAR_Sudu2_Middle:=CANI_VAR38E67;
	END_IF
END_IF
	
IF CANI_IB_VAR16_BOOL_4 AND CANI_IB_VAR48E1 THEN
	IF CANI_VAR48E23<>0 THEN
		PAR_Angle4:=CANI_VAR48E23;
	END_IF
	IF CANI_VAR48E45<>0 THEN
		PAR_Angle5:=CANI_VAR48E45;
	END_IF
	IF CANI_VAR48E67<>0 THEN
		PAR_Angle6:=CANI_VAR48E67;
	END_IF
END_IF
(*阀D加压限压控制*)
IF CANI_IB_VAR17_BOOL AND CANI_IB_VAR18E1 THEN
	IF CANI_VAR18E23<>0 THEN
		PAR_ValveD_PosFull:=CANI_VAR18E23;
	END_IF
	
	IF CANI_VAR18E45<>0 THEN
		PAR_ValveD_NegFull:=CANI_VAR18E45;
	END_IF
END_IF

(*阀C*)
IF CANI_IB_VAR34_BOOL AND CANI_IB_VAR18E1 THEN
	IF CANI_VAR18E23<>0 THEN
		PAR_ValveC_PosFull:=CANI_VAR18E23;
	END_IF
	
	IF CANI_VAR18E45<>0 THEN
		PAR_ValveC_NegFull:=CANI_VAR18E45;
	END_IF
END_IF


(*GPS永久解锁密码*)
IF CANI_IB_VAR30_BOOL AND CANI_IB_VAR18E1 THEN
	IF CANI_VAR18E23<>0 OR CANI_VAR18E45<>0  THEN
		PAR_GPS_ForeverUnlockPassword:=UINT_TO_DINT(CANI_VAR18E23)+65536*UINT_TO_DINT(CANI_VAR18E45);
	END_IF
END_IF

(*泵参数*)
IF NOT CANI_IB_VAR33_BOOL THEN
	CANI_IB_VAR33_BOOL_2:=FALSE;
	CANI_IB_VAR33_BOOL_3:=FALSE;
	CANI_IB_VAR33_BOOL_4:=FALSE;
END_IF
IF CANI_IB_VAR33_BOOL AND CANI_IB_VAR18E1 THEN
	IF CANI_VAR18E23<>0 THEN
		PAR_SpeedLow_Idling:=CANI_VAR18E23;(*低怠速*)
	END_IF
	IF CANI_VAR18E45<>0 THEN
		PAR_SpeedHigh_Idling:=CANI_VAR18E45;(*高怠速*)
	END_IF
	IF CANI_VAR18E67<>0 THEN
		PAR_Y1_PosFull:=CANI_VAR18E67;(*主泵y1最大值*)
	END_IF
END_IF
IF CANI_IB_VAR33_BOOL_2 AND CANI_IB_VAR28E1 THEN
	IF CANI_VAR28E23<>0 THEN
		PAR_Y1_NegFull:=CANI_VAR28E23;(*主泵y1最小值*)
	END_IF
	IF CANI_VAR28E45<>0 THEN
		PAR_Y2_PosFull:=CANI_VAR28E45;(*主泵y2最大值*)
	END_IF
	IF CANI_VAR28E67<>0 THEN
		PAR_Y2_NegFull:=CANI_VAR28E67;(*主泵y2最小值*)
	END_IF
END_IF
IF CANI_IB_VAR33_BOOL_3 AND CANI_IB_VAR38E1 THEN
	IF CANI_VAR38E23<>0 THEN
		PAR_Valve1_PosFull:=CANI_VAR38E23;(*主阀1最大值*)
	END_IF
	IF CANI_VAR38E45<>0 THEN
		PAR_Valve1_NegFull:=CANI_VAR38E45;(*主阀1最小值*)
	END_IF
	IF CANI_VAR38E67<>0 THEN
		PAR_Valve2_PosFull:=CANI_VAR38E67;(*主阀2最大值*)
	END_IF
END_IF
IF CANI_IB_VAR33_BOOL_4 AND CANI_IB_VAR48E1 THEN
	IF CANI_VAR48E23<>0 THEN
		PAR_Valve2_NegFull:=CANI_VAR48E23;(*主阀2最小值*)
	END_IF
	IF CANI_VAR48E45<>0 THEN
		PAR_Valve3_PosFull:=CANI_VAR48E45;(*主阀3最大值*)
	END_IF
	IF CANI_VAR48E67<>0 THEN
		PAR_Valve3_NegFull:=CANI_VAR48E67;(*主阀3最小值*)
	END_IF
END_IF

(*PressAdjust*)
(*IF CANI_IB_VAR34_BOOL AND CANI_IB_VAR18E1 THEN
	IF CANI_VAR18E23<>0 THEN
		PAR_Y21_PosFull:=CANI_VAR18E23;
	END_IF
	IF CANI_VAR18E45<>0 THEN
		PAR_Y21_NegFull:=CANI_VAR18E45;
	END_IF
END_IF*)

(*GPS临时解锁密码*)
IF CANI_IB_VAR36_BOOL AND CANI_IB_VAR18E1 THEN
	IF CANI_VAR18E23<>0 OR CANI_VAR18E45<>0  THEN
		VarGpsTempUnlockPassword:=CANI_VAR18E23;
		VarGpsPasswordTemporaryCode:=CANI_VAR18E23+65536*CANI_VAR18E45;
	END_IF
	
END_IF

(*油门设置界面*)
IF CANI_IB_VAR37_BOOL AND CANI_IB_VAR18E1 THEN
	CANI_Button_YouMen_Min:=BYTE_TO_BOOL(receive_data18E[2] AND 2#00000001);
	CANI_Button_YouMen_Max:=BYTE_TO_BOOL(receive_data18E[3] AND 2#00000001);
	CANI_Button_YouMen_Motor:=BYTE_TO_BOOL(receive_data18E[4] AND 2#00000001);
END_IF
(*桅杆标定界面*)
IF CANI_IB_VAR38_BOOL AND CANI_IB_VAR18E1 THEN
	CANI_Button_L_Limit:=BYTE_TO_BOOL(receive_data18E[2] AND 2#00000001);
	CANI_Button_R_Limit:=BYTE_TO_BOOL(receive_data18E[3] AND 2#00000001);
END_IF

(*液压功能选择界面*)
IF CANI_IB_VAR40_BOOL AND CANI_IB_VAR18E1 THEN
		PAR_MainPumpChioce:=receive_data18E[2];
		PAR_M4ValveChioce:=receive_data18E[3];
		PAR_MotorChioce:=receive_data18E[4];
END_IF

(*加压卷扬设置界面*)
IF CANI_IB_VAR41_BOOL AND CANI_IB_VAR18E1 THEN
(*	IF CANI_VAR18E23<>0 THEN
		PAR_JiYaWinch_Diameter:=CANI_VAR18E23;
	END_IF
	CANI_Button_JiYaWinchDepth_Clear:=BYTE_TO_BOOL(receive_data18E[4] AND 2#00000001);*)
	(*IF CANI_VAR18E23<>0 THEN
		PAR_MainWinchLaLi_Low:=CANI_VAR18E23;
	END_IF*)
	PAR_MainWinchLaLi_Low:=CANI_VAR18E23;
END_IF

(*电比例阀参数设置界面*)
IF NOT CANI_IB_VAR42_BOOL THEN
	CANI_IB_VAR42_BOOL_2:= FALSE;
END_IF

IF CANI_IB_VAR42_BOOL AND CANI_IB_VAR18E1 THEN
	IF CANI_VAR18E23<>0 THEN
		PAR_Y5_PosFull:=CANI_VAR18E23;
	END_IF
	IF CANI_VAR18E45<>0 THEN
		PAR_Y5_NegFull:=CANI_VAR18E45;
	END_IF
	IF CANI_VAR18E67<>0 THEN
		PAR_Y6_PosFull:=CANI_VAR18E67;
	END_IF
END_IF

IF CANI_IB_VAR42_BOOL_2 AND CANI_IB_VAR28E1 THEN
	IF CANI_VAR28E23<>0 THEN
		PAR_Y6_NegFull:=CANI_VAR28E23;
	END_IF
	IF CANI_VAR28E45<>0 THEN
		PAR_Y3_PosFull:=CANI_VAR28E45;
	END_IF
	IF CANI_VAR28E67<>0 THEN
		PAR_Y3_NegFull:=CANI_VAR28E67;
	END_IF
END_IF

IF CANI_IB_VAR42_BOOL_3 AND CANI_IB_VAR38E1 THEN
	IF CANI_VAR38E23<>0 THEN
		PAR_Y4_PosFull:=CANI_VAR38E23;
	END_IF
	IF CANI_VAR38E45<>0 THEN
		PAR_Y4_NegFull:=CANI_VAR38E45;
	END_IF
END_IF

(*节能接收0x18E*)
IF CANI_IB_VAR80_BOOL AND CANI_IB_VAR18E1 THEN
	IF BYTE_TO_BOOL(receive_data18E[2] AND 2#00000001) THEN
		IF NOT SaveEngineState THEN
		SaveEngineState:=TRUE;//节能开
		END_IF
	ELSE
		IF SaveEngineState THEN
		SaveEngineState:=FALSE;	//节能关
		END_IF
	END_IF	
END_IF
IF CANI_IB_VAR80_BOOL AND CANI_IB_VAR18E1 THEN
	IF BYTE_TO_BOOL(receive_data18E[3] AND 2#00000001) THEN
		IF NOT GVL_SaveEngine.AcDecompression THEN
		GVL_SaveEngine.AcDecompression:=TRUE;//泄压开
		END_IF
	ELSE
		IF GVL_SaveEngine.AcDecompression THEN
		GVL_SaveEngine.AcDecompression:=FALSE;	//泄压关
		END_IF
	END_IF
END_IF

//后处理系统
IF CANI_IB_VAR48_BOOL AND CANI_IB_VAR18E1 THEN
	VarZaishengjinzhiSwitch:=BYTE_TO_BOOL(receive_data18E[2] AND 2#00000001);
	VarQiangzhiZaishengSwitch:=BYTE_TO_BOOL(receive_data18E[2] AND 2#00000010);
END_IF


(***********发送************)
//回转角度计算
(*检测回转编码器角度*)
IF PI_Rotation_COUNTER>=0 THEN
	PI_ROTATE_VALUE:=(DINT_TO_UINT(PI_Rotation_COUNTER MOD 2048))*2;
ELSIF  PI_Rotation_COUNTER<0 THEN
	PI_ROTATE_VALUE:=(DINT_TO_UINT(2048+(PI_Rotation_COUNTER MOD 2048)))*2;
END_IF
CANO_R_ANGLE:=REAL_TO_UINT((UINT_TO_REAL(PI_ROTATE_VALUE)/4096)*3600+500);

(*CAN1发送*)
TIME_100ms(IN:=NOT TIME_100ms.Q,PT:=T#100MS);
TIME_200ms(IN:=NOT TIME_200ms.Q,PT:=T#100MS);
TIME_300ms(IN:=NOT TIME_300ms.Q,PT:=T#300MS);
TIME_500ms(IN:=NOT TIME_500ms.Q,PT:=T#500MS);
TIME_700ms(IN:=NOT TIME_700ms.Q,PT:=T#700MS);
TIME_1000ms(IN:=NOT TIME_1000ms.Q,PT:=T#100MS);

send_data187[0]:=UINT_TO_USINT(CANO_ANGLE_X MOD 256);//倾角X
send_data187[1]:=UINT_TO_USINT(CANO_ANGLE_X/256);
send_data187[2]:=UINT_TO_USINT(CANO_ANGLE_Y MOD 256);//倾角Y
send_data187[3]:=UINT_TO_USINT(CANO_ANGLE_Y/256);
send_data187[4]:=UINT_TO_USINT(CANO_R_ANGLE MOD 256);//回转角度
send_data187[5]:=UINT_TO_USINT(CANO_R_ANGLE/256);
send_data187[6]:=UINT_TO_USINT(CANO_Hyd_Tem MOD 256);//液压油温低字节,单位℃
send_data187[7]:=UINT_TO_USINT(CANO_Hyd_Tem/256);
CAN1_SEND_187(xEnable:= TIME_100ms.Q, eChannel:= 0, udiID:= 16#187, xExtended:=FALSE, usiDLC:=8 , aData:=send_data187 );

send_data287[0]:=UdiNT_TO_USINT(PI_SP2A MOD 256);
send_data287[1]:=UdINT_TO_USINT(PI_SP2A/256);
IF(NOT VarGpsSystemLockedState) THEN
	send_data287[2]:=INT_TO_USINT(CANO_water_tem MOD 256);//水温℃
	send_data287[3]:=INT_TO_USINT(CANO_water_tem/256);
	send_data287[4]:=UINT_TO_USINT(CANO_DonglitouPressure MOD 256);//动力头压力
	send_data287[5]:=UINT_TO_USINT(CANO_DonglitouPressure/256);
ELSE
	send_data287[2]:=0;//水温℃
	send_data287[3]:=0;
	send_data287[4]:=0;//动力头压力
	send_data287[5]:=0;
END_IF
send_data287[6]:=UdINT_TO_USINT(PI_SP2B MOD 256);
send_data287[7]:=UdINT_TO_USINT(PI_SP2B/256);
CAN1_SEND_287(xEnable:= TIME_100ms.Q, eChannel:= 0, udiID:= 16#287, xExtended:=FALSE, usiDLC:=8 , aData:=send_data287 );

send_data387[0]:=UINT_TO_USINT(AI_P7 MOD 256);//先导压力传感器端口值
send_data387[1]:=UINT_TO_USINT(AI_P7/256);
send_data387[2]:=UINT_TO_USINT(CANO_DEPTH MOD 256);//当前孔深cm 
send_data387[3]:=UINT_TO_USINT(CANO_DEPTH/256);
send_data387[4]:=UINT_TO_USINT(CANO_FUEL_LEVEL MOD 256);//燃油液位
send_data387[5]:=UINT_TO_USINT(CANO_FUEL_LEVEL/256);
IF(NOT VarGpsSystemLockedState) THEN
	send_data387[6]:=UINT_TO_USINT(CANO_SPEED MOD 256);
	send_data387[7]:=UINT_TO_USINT(CANO_SPEED/256);
ELSE
	send_data387[6]:=0;
	send_data387[7]:=0;
END_IF
//CAN1_SEND_387(xEnable:= TIME_200ms.Q, eChannel:= 0, udiID:= 16#387, xExtended:=FALSE, usiDLC:=8 , aData:=send_data387 );
CAN1_SEND_387(xEnable:= TIME_200ms.Q, eChannel:= 0, udiID:= 16#387, xExtended:=FALSE, usiDLC:=8 , aData:=send_data387 );

//电瓶电压报警
IF(CANO_VOL_VALUE<25000)THEN
	CANO_TooLow_BatteryVol:=TRUE;
ELSE
	CANO_TooLow_BatteryVol:=FALSE;
END_IF
//主卷上限位报警
IF(DIL_SQ4 OR (NOT DIH_SQ8)) THEN
	CANO_UpLimitWarn:=TRUE;
ELSE
	CANO_UpLimitWarn:=FALSE;
END_IF

send_data487[0]:=PACK(B0:=0,B1:=CANO_TooLow_BatteryVol,B2:=TRUE,(*B2:=DIL_SQ13,*)B3:=CANO_RotationModle ,
					  B4:=CANO_TooLow_FUEL_LEVEL,B5:=DOH_Y51,B6:=CANO_UpLimitWarn,B7:=(DOH_Y56 AND DOH_Y55));
send_data487[1]:=PACK(B0:=CANO_TooHigh_HydOilTem,B1:=CANO_TooLow_OilPress,B2:=CANO_TooHigh_WaterTem,B3:=VarMastAutoEnable ,
					  B4:=DIH_SP4,B5:=0,B6:=VarMastLimitCancel,B7:=0);
IF(NOT VarGpsSystemLockedState) THEN
	send_data487[2]:=UINT_TO_USINT(CANO_JiayaPressure MOD 256); //加压压力
	send_data487[3]:=UINT_TO_USINT(CANO_JiayaPressure/256);
	send_data487[4]:=UINT_TO_USINT(CANO_ZhuJuanPressure MOD 256);//主卷压力
	send_data487[5]:=UINT_TO_USINT(CANO_ZhuJuanPressure/256);
	send_data487[6]:=UINT_TO_USINT(CANO_Lub_Press MOD 256);
	send_data487[7]:=UINT_TO_USINT(CANO_Lub_Press/256);
ELSE
	send_data487[2]:=UINT_TO_USINT(0 MOD 256); //加压压力
	send_data487[3]:=UINT_TO_USINT(0/256);
	send_data487[4]:=UINT_TO_USINT(0 MOD 256);//主卷压力
	send_data487[5]:=UINT_TO_USINT(0/256);
	send_data487[6]:=UINT_TO_USINT(0 MOD 256);//发动机机油压力
	send_data487[7]:=UINT_TO_USINT(0/256);
END_IF
CAN1_SEND_487(xEnable:= TIME_200ms.Q, eChannel:= 0, udiID:= 16#487, xExtended:=FALSE, usiDLC:=8 , aData:=send_data487 );

send_data188[0]:=DINT_TO_USINT(PI_Rotation_COUNTER MOD 256); //回转PI
send_data188[1]:=DINT_TO_USINT(PI_Rotation_COUNTER/256);
send_data188[2]:=UINT_TO_USINT(AI_P1 MOD 256);//推进压力端口值P1
send_data188[3]:=UINT_TO_USINT(AI_P1/256);
send_data188[4]:=UINT_TO_USINT(AI_SP1 MOD 256);//燃油液位端口值SP1
send_data188[5]:=UINT_TO_USINT(AI_SP1/256);
send_data188[6]:=UINT_TO_USINT(PWM_Y29 MOD 256); //右油缸伸
send_data188[7]:=UINT_TO_USINT(PWM_Y29/256);
CAN1_SEND_188(xEnable:= TIME_1000ms.Q, eChannel:= 0, udiID:= 16#188, xExtended:=FALSE, usiDLC:=8 , aData:=send_data188 );

(*GPS总线故障报警*)
send_data288[0]:=PACK(B0:=CANO_SensorError_Joy,B1:=CANO_SensorError_Angle,B2:=CANO_SensorError_Rotation,B3:=CANO_SensorError_DonglitouPress ,
					  B4:=0,B5:=CANO_SensorError_HydOilTem,B6:=CANO_SensorError_JiaYaPress,B7:=CANO_SensorError_ZhuJuanPress);
send_data288[1]:=PACK(B0:=CANO_SensorError_FuelLevel,B1:=0,B2:=0,B3:=(VarCanGpsTongXunLockCommand OR VarCanGpsFakeLockCommand) AND VarGpsSystemLockedState,
					  B4:=0,B5:=DIH_SQ1,B6:=DIH_SQ2,B7:=VarCanGpsTongXunLockCommand AND VarGpsSystemLockedState);
send_data288[2]:=UINT_TO_USINT(PWM_Y27 MOD 256);//左油缸伸
send_data288[3]:=UINT_TO_USINT(PWM_Y27/256);
send_data288[4]:=UINT_TO_USINT(PWM_Y28 MOD 256);//左油缸缩
send_data288[5]:=UINT_TO_USINT(PWM_Y28/256);
send_data288[6]:=UINT_TO_USINT(PWM_Y30 MOD 256);//右油缸缩
send_data288[7]:=UINT_TO_USINT(PWM_Y30/256);
CAN1_SEND_288(xEnable:= TIME_1000ms.Q, eChannel:= 0, udiID:= 16#288, xExtended:=FALSE, usiDLC:=8 , aData:=send_data288 );


send_data388[0]:=PACK(B0:=DIL_SQ11,B1:=DIH_SQ12,B2:=0,B3:=0,
					  B4:=0,B5:=0,B6:=0,B7:=0);
send_data388[1]:=PACK(B0:=DIL_SQ4,B1:=DIH_SP4,B2:=DIH_JOY,B3:=DIH_SA8,
					  B4:=DIL_SQ3,B5:=DIH_SQ5,B6:=DIH_SQ6,B7:=DIH_SQ8);
send_data388[2]:=UINT_TO_USINT(AI_SP7 MOD 256);
send_data388[3]:=UINT_TO_USINT(AI_SP7/256);
send_data388[4]:=UINT_TO_USINT(CANO_PowerHeadTorque MOD 256);
send_data388[5]:=UINT_TO_USINT(CANO_PowerHeadTorque/256);
send_data388[6]:=DINT_TO_USINT(PI_Rotation_COUNTER MOD 256);
send_data388[7]:=DINT_TO_USINT(PI_Rotation_COUNTER/256);
CAN1_SEND_388(xEnable:= TIME_1000ms.Q, eChannel:= 0, udiID:= 16#388, xExtended:=FALSE, usiDLC:=8 , aData:=send_data388 );

send_data488[0]:=UINT_TO_USINT(PWM_Y21 MOD 256);// 左回转
send_data488[1]:=UINT_TO_USINT(PWM_Y21/256);
send_data488[2]:=UINT_TO_USINT(PWM_Y22 MOD 256);// 右回转
send_data488[3]:=UINT_TO_USINT(PWM_Y22/256);
send_data488[4]:=UINT_TO_USINT((CANO_VOL_VALUE/10) MOD 256);//电压
send_data488[5]:=UINT_TO_USINT((CANO_VOL_VALUE/10)/256);
send_data488[6]:=UINT_TO_USINT(CANO_PowerHeadSpeed MOD 256);
send_data488[7]:=UINT_TO_USINT(CANO_PowerHeadSpeed/256);
CAN1_SEND_488(xEnable:= TIME_1000ms.Q, eChannel:= 0, udiID:= 16#488, xExtended:=FALSE, usiDLC:=8 , aData:=send_data488 );

send_data189[0]:=UINT_TO_USINT(AI_P3 MOD 256);
send_data189[1]:=UINT_TO_USINT(AI_P3/256);
send_data189[2]:=UINT_TO_USINT(AI_P2 MOD 256);
send_data189[3]:=UINT_TO_USINT(AI_P2/256);
send_data189[4]:=UINT_TO_USINT(AI_JOYX MOD 256);
send_data189[5]:=UINT_TO_USINT(AI_JOYX/256);
send_data189[6]:=UINT_TO_USINT(AI_JOYY MOD 256);
send_data189[7]:=UINT_TO_USINT(AI_JOYY/256);
CAN1_SEND_189(xEnable:= TIME_1000ms.Q, eChannel:= 0, udiID:= 16#189, xExtended:=FALSE, usiDLC:=8 , aData:=send_data189);

send_data289[0]:=UINT_TO_USINT(PWM_Y1 MOD 256);
send_data289[1]:=UINT_TO_USINT(PWM_Y1/256);
send_data289[2]:=DINT_TO_USINT(CANO_engine_hour_h MOD 256);
send_data289[3]:=DINT_TO_USINT(CANO_engine_hour_h/256);
send_data289[4]:=UINT_TO_USINT(CANO_engine_hour_m MOD 256);
send_data289[5]:=UINT_TO_USINT(CANO_engine_hour_m/256);
send_data289[6]:=UINT_TO_USINT(PWM_Y2 MOD 256);
send_data289[7]:=UINT_TO_USINT(PWM_Y2/256);
//CAN1_SEND_289(xEnable:= TIME_200ms.Q, eChannel:= 0, udiID:= 16#289, xExtended:=FALSE, usiDLC:=8 , aData:=send_data289);
CAN1_SEND_289(xEnable:= TRUE, eChannel:= 0, udiID:= 16#289, xExtended:=FALSE, usiDLC:=8 , aData:=send_data289);

send_data389[0]:=UINT_TO_USINT(PWM_Y3 MOD 256);
send_data389[1]:=UINT_TO_USINT(PWM_Y3/256);
send_data389[2]:=UINT_TO_USINT(PWM_Y4 MOD 256);
send_data389[3]:=UINT_TO_USINT(PWM_Y4/256);
send_data389[4]:=UINT_TO_USINT(AI_SP3 MOD 256);
send_data389[5]:=UINT_TO_USINT(AI_SP3/256);
send_data389[6]:=UINT_TO_USINT(PWM_Y34 MOD 256);
send_data389[7]:=UINT_TO_USINT(PWM_Y34/256);
CAN1_SEND_389(xEnable:= TIME_1000ms.Q, eChannel:= 0, udiID:= 16#389, xExtended:=FALSE, usiDLC:=8 , aData:=send_data389);

send_data489[0]:=UINT_TO_USINT(PWM_Y5 MOD 256);
send_data489[1]:=UINT_TO_USINT(PWM_Y5/256);
send_data489[2]:=PACK(B0:=((VarCanGpsTongXunLockCommand OR VarCanGpsFakeLockCommand) AND VarGpsGlobalEnable) ,B1:=0,B2:=0,
						B3:=(VarCanGpsKongZhiQiLockCommand AND VarGpsGlobalEnable),
					    B4:=0,B5:=(VarCanGpsYanShiLockCommand AND VarGpsGlobalEnable),
						B6:=(VarCanGpsTianXianLockCommand AND VarGpsGlobalEnable ),
 						B7:=(VarCanGpsKaiGaiLockCommand AND VarGpsGlobalEnable));
send_data489[3]:=UINT_TO_USINT(0);
send_data489[4]:=UDINT_TO_USINT((CANO_Accumu_Fuel MOD 65536) MOD 256);
send_data489[5]:=UDINT_TO_USINT((CANO_Accumu_Fuel MOD 65536)/256);
send_data489[6]:=UDINT_TO_USINT((CANO_Accumu_Fuel/65536) MOD 256);
send_data489[7]:=UDINT_TO_USINT((CANO_Accumu_Fuel/65536) /256);
CAN1_SEND_489(xEnable:= TIME_1000ms.Q, eChannel:= 0, udiID:= 16#489, xExtended:=FALSE, usiDLC:=8 , aData:=send_data489);

send_data18A[0]:=UDINT_TO_USINT((CANO_ACCMUDEPTH/100 MOD 65536) MOD 256);
send_data18A[1]:=UDINT_TO_USINT((CANO_ACCMUDEPTH/100 MOD 65536)/256);
send_data18A[2]:=UDINT_TO_USINT((CANO_ACCMUDEPTH/100 /65536) MOD 256);
send_data18A[3]:=UDINT_TO_USINT((CANO_ACCMUDEPTH/100 /65536)/256);
send_data18A[4]:=UINT_TO_USINT(CANO_LimiteModle MOD 256);
send_data18A[5]:=UINT_TO_USINT(CANO_LimiteModle/256);
send_data18A[6]:=UINT_TO_USINT(0 MOD 256);
send_data18A[7]:=UINT_TO_USINT(0/256);
CAN1_SEND_18A(xEnable:= TIME_1000ms.Q, eChannel:= 0, udiID:= 16#18A, xExtended:=FALSE, usiDLC:=8 , aData:=send_data18A);

send_data28A[0]:=UINT_TO_USINT(PAR_Circle1 MOD 256);
send_data28A[1]:=UINT_TO_USINT(PAR_Circle1/256);
send_data28A[2]:=UINT_TO_USINT(PAR_Circle2 MOD 256);
send_data28A[3]:=UINT_TO_USINT(PAR_Circle2/256);
send_data28A[4]:=UINT_TO_USINT(PAR_Quanshu MOD 256);
send_data28A[5]:=UINT_TO_USINT(PAR_Quanshu/256);
send_data28A[6]:=UINT_TO_USINT(PAR_Sudu1_Min MOD 256);
send_data28A[7]:=UINT_TO_USINT(PAR_Sudu1_Min/256);
CAN1_SEND_28A(xEnable:= TIME_200ms.Q, eChannel:= 0, udiID:= 16#28A, xExtended:=FALSE, usiDLC:=8 , aData:=send_data28A);

send_data38A[0]:=UINT_TO_USINT(PAR_Sudu1_Max MOD 256);
send_data38A[1]:=UINT_TO_USINT(PAR_Sudu1_Max/256);
send_data38A[2]:=UINT_TO_USINT(PAR_Sudu1_Middle MOD 256);
send_data38A[3]:=UINT_TO_USINT(PAR_Sudu1_Middle/256);
send_data38A[4]:=UINT_TO_USINT(PAR_Angle1 MOD 256);
send_data38A[5]:=UINT_TO_USINT(PAR_Angle1/256);
send_data38A[6]:=UINT_TO_USINT(PAR_Angle2 MOD 256);
send_data38A[7]:=UINT_TO_USINT(PAR_Angle2/256);
CAN1_SEND_38A(xEnable:= TIME_1000ms.Q, eChannel:= 0, udiID:= 16#38A, xExtended:=FALSE, usiDLC:=8 , aData:=send_data38A);

send_data48A[0]:=UINT_TO_USINT(PAR_Angle3 MOD 256);
send_data48A[1]:=UINT_TO_USINT(PAR_Angle3/256);
send_data48A[2]:=UINT_TO_USINT(PAR_Sudu2_Min MOD 256);
send_data48A[3]:=UINT_TO_USINT(PAR_Sudu2_Min/256);
send_data48A[4]:=UINT_TO_USINT(PAR_Sudu2_Max MOD 256);
send_data48A[5]:=UINT_TO_USINT(PAR_Sudu2_Max/256);
send_data48A[6]:=UINT_TO_USINT(PAR_Sudu2_Middle MOD 256);
send_data48A[7]:=UINT_TO_USINT(PAR_Sudu2_Middle/256);
CAN1_SEND_48A(xEnable:= TIME_1000ms.Q, eChannel:= 0, udiID:= 16#48A, xExtended:=FALSE, usiDLC:=8 , aData:=send_data48A);

send_data18B[0]:=UINT_TO_USINT(PAR_Angle4 MOD 256);
send_data18B[1]:=UINT_TO_USINT(PAR_Angle4/256);
send_data18B[2]:=UINT_TO_USINT(PAR_Angle5 MOD 256);
send_data18B[3]:=UINT_TO_USINT(PAR_Angle5/256);
send_data18B[4]:=UINT_TO_USINT(PAR_Angle6 MOD 256);
send_data18B[5]:=UINT_TO_USINT(PAR_Angle6/256);
send_data18B[6]:=UINT_TO_USINT(AI_ECM2_9 MOD 256);
send_data18B[7]:=UINT_TO_USINT(AI_ECM2_9/256);
CAN1_SEND_18B(xEnable:= TIME_1000ms.Q, eChannel:= 0, udiID:= 16#18B, xExtended:=FALSE, usiDLC:=8 , aData:=send_data18B);

send_data28B[0]:=UINT_TO_USINT(PAR_YouMen_NegFull MOD 256);
send_data28B[1]:=UINT_TO_USINT(PAR_YouMen_NegFull/256);
send_data28B[2]:=UINT_TO_USINT(PAR_YouMen_PosFull MOD 256);
send_data28B[3]:=UINT_TO_USINT(PAR_YouMen_PosFull/256);
send_data28B[4]:=UINT_TO_USINT(PAR_Y27_PosFull MOD 256);
send_data28B[5]:=UINT_TO_USINT(PAR_Y27_PosFull/256);
send_data28B[6]:=UINT_TO_USINT(PAR_Y27_NegFull MOD 256);
send_data28B[7]:=UINT_TO_USINT(PAR_Y27_NegFull/256);
CAN1_SEND_28B(xEnable:= TIME_1000ms.Q, eChannel:= 0, udiID:= 16#28B, xExtended:=FALSE, usiDLC:=8 , aData:=send_data28B);

send_data38B[0]:=UINT_TO_USINT(PAR_Y28_PosFull MOD 256);
send_data38B[1]:=UINT_TO_USINT(PAR_Y28_PosFull/256);
send_data38B[2]:=UINT_TO_USINT(PAR_Y28_NegFull MOD 256);
send_data38B[3]:=UINT_TO_USINT(PAR_Y28_NegFull/256);
send_data38B[4]:=UINT_TO_USINT(PAR_Y29_PosFull MOD 256);
send_data38B[5]:=UINT_TO_USINT(PAR_Y29_PosFull/256);
send_data38B[6]:=UINT_TO_USINT(PAR_Y29_NegFull MOD 256);
send_data38B[7]:=UINT_TO_USINT(PAR_Y29_NegFull/256);
CAN1_SEND_38B(xEnable:= TIME_1000ms.Q, eChannel:= 0, udiID:= 16#38B, xExtended:=FALSE, usiDLC:=8 , aData:=send_data38B);

send_data48B[0]:=UINT_TO_USINT(PAR_Y30_PosFull MOD 256);
send_data48B[1]:=UINT_TO_USINT(PAR_Y30_PosFull/256);
send_data48B[2]:=UINT_TO_USINT(PAR_Y30_NegFull MOD 256);
send_data48B[3]:=UINT_TO_USINT(PAR_Y30_NegFull/256);
send_data48B[4]:=UINT_TO_USINT(PAR_L_LimiteValue MOD 256);
send_data48B[5]:=UINT_TO_USINT(PAR_L_LimiteValue/256);
send_data48B[6]:=UINT_TO_USINT(PAR_R_LimiteValue MOD 256);
send_data48B[7]:=UINT_TO_USINT(PAR_R_LimiteValue/256);
CAN1_SEND_48B(xEnable:= TIME_1000ms.Q, eChannel:= 0, udiID:= 16#48B, xExtended:=FALSE, usiDLC:=8 , aData:=send_data48B);

send_data18C[0]:=UINT_TO_USINT(AI_SP11 MOD 256);
send_data18C[1]:=UINT_TO_USINT(AI_SP11/256);
send_data18C[2]:=UINT_TO_USINT(PWM_Y6 MOD 256);
send_data18C[3]:=UINT_TO_USINT(PWM_Y6/256);
send_data18C[4]:=UINT_TO_USINT(CANO_RotationStop_Pressure MOD 256);
send_data18C[5]:=UINT_TO_USINT(CANO_RotationStop_Pressure/256);
send_data18C[6]:=UINT_TO_USINT(PWM_Y7 MOD 256);
send_data18C[7]:=UINT_TO_USINT(PWM_Y7/256);
CAN1_SEND_18C(xEnable:= TIME_1000ms.Q, eChannel:= 0, udiID:= 16#18C, xExtended:=FALSE, usiDLC:=8 , aData:=send_data18C);

send_data28C[0]:=UINT_TO_USINT(PWM_Y8 MOD 256);
send_data28C[1]:=UINT_TO_USINT(PWM_Y8/256);
send_data28C[2]:=UINT_TO_USINT(AI_P8 MOD 256);
send_data28C[3]:=UINT_TO_USINT(AI_P8/256);
send_data28C[4]:=UINT_TO_USINT(PWM_Y9 MOD 256);
send_data28C[5]:=UINT_TO_USINT(PWM_Y9/256);
send_data28C[6]:=UINT_TO_USINT(CANO_PilotPressure MOD 256);
send_data28C[7]:=UINT_TO_USINT(CANO_PilotPressure/256);
CAN1_SEND_28C(xEnable:= TIME_1000ms.Q, eChannel:= 0, udiID:= 16#28C, xExtended:=FALSE, usiDLC:=8 , aData:=send_data28C);

send_data38C[0]:=UDINT_TO_USINT((Codes_SPN_1 MOD 65536) MOD 256);
send_data38C[1]:=UDINT_TO_USINT((Codes_SPN_1 MOD 65536)/256);
send_data38C[2]:=UDINT_TO_USINT((Codes_SPN_1/65536) MOD 256);
send_data38C[3]:=UDINT_TO_USINT((Codes_SPN_1/65536)/256);
send_data38C[4]:=UDINT_TO_USINT((Codes_SPN_2 MOD 65536) MOD 256);
send_data38C[5]:=UDINT_TO_USINT((Codes_SPN_2 MOD 65536)/256);
send_data38C[6]:=UDINT_TO_USINT((Codes_SPN_2/65536) MOD 256);
send_data38C[7]:=UDINT_TO_USINT((Codes_SPN_2/65536)/256);
CAN1_SEND_38C(xEnable:= TIME_1000ms.Q, eChannel:= 0, udiID:= 16#38C, xExtended:=FALSE, usiDLC:=8 , aData:=send_data38C);

send_data48C[0]:=UDINT_TO_USINT((Codes_SPN_3 MOD 65536) MOD 256);
send_data48C[1]:=UDINT_TO_USINT((Codes_SPN_3 MOD 65536)/256);
send_data48C[2]:=UDINT_TO_USINT((Codes_SPN_3/65536) MOD 256);
send_data48C[3]:=UDINT_TO_USINT((Codes_SPN_3/65536)/256);
send_data48C[4]:=UDINT_TO_USINT((Codes_SPN_4 MOD 65536) MOD 256);
send_data48C[5]:=UDINT_TO_USINT((Codes_SPN_4 MOD 65536)/256);
send_data48C[6]:=UDINT_TO_USINT((Codes_SPN_4/65536) MOD 256);
send_data48C[7]:=UDINT_TO_USINT((Codes_SPN_4/65536)/256);
CAN1_SEND_48C(xEnable:= TIME_1000ms.Q, eChannel:= 0, udiID:= 16#48C, xExtended:=FALSE, usiDLC:=8 , aData:=send_data48C);

send_data18D[0]:=UINT_TO_USINT(FuelMomentary MOD 256);
send_data18D[1]:=UINT_TO_USINT(FuelMomentary/256);
send_data18D[2]:=UINT_TO_USINT((REAL_TO_UINT(Pressure_Coe*100)) MOD 256);
send_data18D[3]:=UINT_TO_USINT((REAL_TO_UINT(Pressure_Coe*100))/256);
send_data18D[4]:=UINT_TO_USINT(CANO_MainWinch_Speed MOD 256);
send_data18D[5]:=UINT_TO_USINT(CANO_MainWinch_Speed/256);
send_data18D[6]:=UINT_TO_USINT(PWM_Y10 MOD 256);
send_data18D[7]:=UINT_TO_USINT(PWM_Y10/256);
CAN1_SEND_18D(xEnable:= TRUE, eChannel:= 0, udiID:= 16#18D, xExtended:=FALSE, usiDLC:=8 , aData:=send_data18D);

send_data28D[0]:=UINT_TO_USINT(0 MOD 256);
send_data28D[1]:=UINT_TO_USINT(0/256);
send_data28D[2]:=UINT_TO_USINT(0 MOD 256);
send_data28D[3]:=UINT_TO_USINT(0/256);
send_data28D[4]:=UINT_TO_USINT(PWM_Y11 MOD 256);
send_data28D[5]:=UINT_TO_USINT(PWM_Y11/256);
send_data28D[6]:=UINT_TO_USINT(PWM_Y12 MOD 256);
send_data28D[7]:=UINT_TO_USINT(PWM_Y12/256);
CAN1_SEND_28D(xEnable:= TIME_1000ms.Q, eChannel:= 0, udiID:= 16#28D, xExtended:=FALSE, usiDLC:=8 , aData:=send_data28D);

send_data38D[0]:=UINT_TO_USINT(0 MOD 256);
send_data38D[1]:=UINT_TO_USINT(0/256);
send_data38D[2]:=UINT_TO_USINT(0 MOD 256);
send_data38D[3]:=UINT_TO_USINT(0/256);
send_data38D[4]:=UINT_TO_USINT(PWM_Y11 MOD 256);
send_data38D[5]:=UINT_TO_USINT(PWM_Y11/256);
send_data38D[6]:=UINT_TO_USINT(PWM_Y12 MOD 256);
send_data38D[7]:=UINT_TO_USINT(PWM_Y12/256);
CAN1_SEND_38D(xEnable:= TIME_1000ms.Q, eChannel:= 0, udiID:= 16#38D, xExtended:=FALSE, usiDLC:=8 , aData:=send_data38D);

send_data48D[0]:=UDINT_TO_USINT((Codes_SPN_5 MOD 65536) MOD 256);
send_data48D[1]:=UDINT_TO_USINT((Codes_SPN_5 MOD 65536)/256);
send_data48D[2]:=UDINT_TO_USINT((Codes_SPN_5/65536) MOD 256);
send_data48D[3]:=UDINT_TO_USINT((Codes_SPN_5/65536)/256);
send_data48D[4]:=UDINT_TO_USINT((Codes_SPN_6 MOD 65536) MOD 256);
send_data48D[5]:=UDINT_TO_USINT((Codes_SPN_6 MOD 65536)/256);
send_data48D[6]:=UDINT_TO_USINT((Codes_SPN_6/65536) MOD 256);
send_data48D[7]:=UDINT_TO_USINT((Codes_SPN_6/65536)/256);
CAN1_SEND_48D(xEnable:= TIME_1000ms.Q, eChannel:= 0, udiID:= 16#48D, xExtended:=FALSE, usiDLC:=8 , aData:=send_data48D);

send_data186[0]:=UDINT_TO_USINT((Codes_SPN_7 MOD 65536) MOD 256);
send_data186[1]:=UDINT_TO_USINT((Codes_SPN_7 MOD 65536)/256);
send_data186[2]:=UDINT_TO_USINT((Codes_SPN_7/65536) MOD 256);
send_data186[3]:=UDINT_TO_USINT((Codes_SPN_7/65536)/256);
send_data186[4]:=UDINT_TO_USINT((Codes_SPN_8 MOD 65536) MOD 256);
send_data186[5]:=UDINT_TO_USINT((Codes_SPN_8 MOD 65536)/256);
send_data186[6]:=UDINT_TO_USINT((Codes_SPN_8/65536) MOD 256);
send_data186[7]:=UDINT_TO_USINT((Codes_SPN_8/65536)/256);
CAN1_SEND_186(xEnable:= TIME_1000ms.Q, eChannel:= 0, udiID:= 16#186, xExtended:=FALSE, usiDLC:=8 , aData:=send_data186);

send_data286[0]:=UDINT_TO_USINT((Codes_SPN_9 MOD 65536) MOD 256);
send_data286[1]:=UDINT_TO_USINT((Codes_SPN_9 MOD 65536)/256);
send_data286[2]:=UDINT_TO_USINT((Codes_SPN_9/65536) MOD 256);
send_data286[3]:=UDINT_TO_USINT((Codes_SPN_9/65536)/256);
send_data286[4]:=UDINT_TO_USINT((Codes_SPN_10 MOD 65536) MOD 256);
send_data286[5]:=UDINT_TO_USINT((Codes_SPN_10 MOD 65536)/256);
send_data286[6]:=UDINT_TO_USINT((Codes_SPN_10/65536) MOD 256);
send_data286[7]:=UDINT_TO_USINT((Codes_SPN_10/65536)/256);
CAN1_SEND_286(xEnable:= TIME_1000ms.Q, eChannel:= 0, udiID:= 16#286, xExtended:=FALSE, usiDLC:=8 , aData:=send_data286);

send_data386[0]:=BYTE_TO_USINT(Codes_FMI_1);
send_data386[1]:=BYTE_TO_USINT(Codes_FMI_2);
send_data386[2]:=BYTE_TO_USINT(Codes_FMI_3);
send_data386[3]:=BYTE_TO_USINT(Codes_FMI_4);
send_data386[4]:=BYTE_TO_USINT(Codes_FMI_5);
send_data386[5]:=BYTE_TO_USINT(Codes_FMI_6);
send_data386[6]:=BYTE_TO_USINT(Codes_FMI_7);
send_data386[7]:=BYTE_TO_USINT(Codes_FMI_8);
CAN1_SEND_386(xEnable:= TIME_1000ms.Q, eChannel:= 0, udiID:= 16#386, xExtended:=FALSE, usiDLC:=8 , aData:=send_data386);

send_data486[0]:=BYTE_TO_USINT(Codes_FMI_9);
send_data486[1]:=BYTE_TO_USINT(Codes_FMI_10);
send_data486[2]:=PACK(B0:=CANO_SensorError_Tension,B1:=CANO_SensorError_PoiltPress,B2:=0,B3:=0,
					  B4:=0,B5:=0,B6:=0,B7:=0);
send_data486[3]:=BYTE_TO_USINT(Codes_FMI_1);
send_data486[4]:=UINT_TO_USINT(PWM_Y13 MOD 256);
send_data486[5]:=UINT_TO_USINT(PWM_Y13/256);
send_data486[6]:=UINT_TO_USINT(PWM_Y14 MOD 256);
send_data486[7]:=UINT_TO_USINT(PWM_Y14/256);
CAN1_SEND_486(xEnable:= TIME_1000ms.Q, eChannel:= 0, udiID:= 16#486, xExtended:=FALSE, usiDLC:=8 , aData:=send_data486);

send_data185[0]:=UINT_TO_USINT(PWM_Y15 MOD 256);
send_data185[1]:=UINT_TO_USINT(PWM_Y15/256);
send_data185[2]:=UINT_TO_USINT(PWM_Y16 MOD 256);
send_data185[3]:=UINT_TO_USINT(PWM_Y16/256);
send_data185[4]:=UINT_TO_USINT(PWM_Y17 MOD 256);
send_data185[5]:=UINT_TO_USINT(PWM_Y17/256);
send_data185[6]:=UINT_TO_USINT(PWM_Y18 MOD 256);
send_data185[7]:=UINT_TO_USINT(PWM_Y18/256);
CAN1_SEND_185(xEnable:= TIME_1000ms.Q, eChannel:= 0, udiID:= 16#185, xExtended:=FALSE, usiDLC:=8 , aData:=send_data185);

send_data285[0]:=UINT_TO_USINT(100 MOD 256);
send_data285[1]:=UINT_TO_USINT(100/256);
send_data285[2]:=UINT_TO_USINT(101 MOD 256);
send_data285[3]:=UINT_TO_USINT(101/256);
send_data285[4]:=UINT_TO_USINT(100 MOD 256);
send_data285[5]:=UINT_TO_USINT(100/256);
send_data285[6]:=UINT_TO_USINT(100 MOD 256);
send_data285[7]:=UINT_TO_USINT(100/256);
CAN1_SEND_285(xEnable:= TIME_1000ms.Q, eChannel:= 0, udiID:= 16#285, xExtended:=FALSE, usiDLC:=8 , aData:=send_data285);

send_data385[0]:=UINT_TO_USINT(0 MOD 256);
send_data385[1]:=UINT_TO_USINT(0/256);
send_data385[2]:=UINT_TO_USINT(0 MOD 256);
send_data385[3]:=UINT_TO_USINT(0/256);
send_data385[4]:=UINT_TO_USINT(PWM_Y19 MOD 256);
send_data385[5]:=UINT_TO_USINT(PWM_Y19/256);
send_data385[6]:=UINT_TO_USINT(PWM_Y20 MOD 256);
send_data385[7]:=UINT_TO_USINT(PWM_Y20/256);
CAN1_SEND_385(xEnable:= TIME_1000ms.Q, eChannel:= 0, udiID:= 16#385, xExtended:=FALSE, usiDLC:=8 , aData:=send_data385);

send_data485[0]:=BOOL_TO_USINT(VarGpsTempUnlockDoing);
send_data485[1]:=UINT_TO_USINT(0/256);
send_data485[2]:=BOOL_TO_USINT(VarGpsGlobalEnable);
send_data485[3]:=UINT_TO_USINT(0/256);
send_data485[4]:=UINT_TO_USINT(0 MOD 256);
send_data485[5]:=UINT_TO_USINT(0/256);
send_data485[6]:=UINT_TO_USINT(0 MOD 256);
send_data485[7]:=UINT_TO_USINT(0/256);
CAN1_SEND_485(xEnable:= TIME_1000ms.Q, eChannel:= 0, udiID:= 16#485, xExtended:=FALSE, usiDLC:=8 , aData:=send_data485);

send_data585[0]:=UINT_TO_USINT(0 MOD 256);
send_data585[1]:=UINT_TO_USINT(0/256);
send_data585[2]:=UINT_TO_USINT(0 MOD 256);
send_data585[3]:=UINT_TO_USINT(0/256);
send_data585[4]:=UINT_TO_USINT(0 MOD 256);
send_data585[5]:=UINT_TO_USINT(0/256);
send_data585[6]:=UINT_TO_USINT(0 MOD 256);
send_data585[7]:=UINT_TO_USINT(0/256);
CAN1_SEND_585(xEnable:= TIME_1000ms.Q, eChannel:= 0, udiID:= 16#585, xExtended:=FALSE, usiDLC:=8 , aData:=send_data585);

send_data685[0]:=UINT_TO_USINT(PWM_Y21 MOD 256);
send_data685[1]:=UINT_TO_USINT(PWM_Y21/256);
send_data685[2]:=UINT_TO_USINT(PWM_Y22 MOD 256);
send_data685[3]:=UINT_TO_USINT(PWM_Y22/256);
send_data685[4]:=UINT_TO_USINT(PAR_SpeedHigh_Idling MOD 256);
send_data685[5]:=UINT_TO_USINT(PAR_SpeedHigh_Idling/256);
send_data685[6]:=UINT_TO_USINT(PAR_SpeedLow_Idling MOD 256);
send_data685[7]:=UINT_TO_USINT(PAR_SpeedLow_Idling/256);
CAN1_SEND_685(xEnable:= TIME_1000ms.Q, eChannel:= 0, udiID:= 16#685, xExtended:=FALSE, usiDLC:=8 , aData:=send_data685);

send_data785[0]:=UINT_TO_USINT(PWM_Y23 MOD 256);
send_data785[1]:=UINT_TO_USINT(PWM_Y23/256);
send_data785[2]:=UINT_TO_USINT(PWM_Y24 MOD 256);
send_data785[3]:=UINT_TO_USINT(PWM_Y24/256);
send_data785[4]:=UINT_TO_USINT(PAR_Y1_PosFull MOD 256);
send_data785[5]:=UINT_TO_USINT(PAR_Y1_PosFull/256);
send_data785[6]:=UINT_TO_USINT(PAR_Y1_NegFull MOD 256);
send_data785[7]:=UINT_TO_USINT(PAR_Y1_NegFull/256);
CAN1_SEND_785(xEnable:= TIME_1000ms.Q, eChannel:= 0, udiID:= 16#785, xExtended:=FALSE, usiDLC:=8 , aData:=send_data785);

send_data184[0]:=UINT_TO_USINT(PWM_Y25 MOD 256);
send_data184[1]:=UINT_TO_USINT(PWM_Y25/256);
send_data184[2]:=UINT_TO_USINT(PWM_Y26 MOD 256);
send_data184[3]:=UINT_TO_USINT(PWM_Y26/256);
send_data184[4]:=UINT_TO_USINT(PWM_Y31 MOD 256);
send_data184[5]:=UINT_TO_USINT(PWM_Y31/256);
send_data184[6]:=UINT_TO_USINT(PWM_Y32 MOD 256);
send_data184[7]:=UINT_TO_USINT(PWM_Y32/256);
CAN1_SEND_184(xEnable:= TIME_1000ms.Q, eChannel:= 0, udiID:= 16#184, xExtended:=FALSE, usiDLC:=8 , aData:=send_data184);

send_data284[0]:=UINT_TO_USINT(PWM_Y33 MOD 256);
send_data284[1]:=UINT_TO_USINT(PWM_Y33/256);
send_data284[2]:=UINT_TO_USINT(PWM_Y35 MOD 256);
send_data284[3]:=UINT_TO_USINT(PWM_Y35/256);
send_data284[4]:=UINT_TO_USINT(PWM_Y37 MOD 256);
send_data284[5]:=UINT_TO_USINT(PWM_Y37/256);
send_data284[6]:=UINT_TO_USINT(PWM_Y38 MOD 256);
send_data284[7]:=UINT_TO_USINT(PWM_Y38/256);
//CAN1_SEND_284(xEnable:= TIME_1000ms.Q, eChannel:= 0, udiID:= 16#284, xExtended:=FALSE, usiDLC:=8 , aData:=send_data284);
CAN1_SEND_284(xEnable:= TRUE, eChannel:= 0, udiID:= 16#284, xExtended:=FALSE, usiDLC:=8 , aData:=send_data284);

send_data384[0]:=UINT_TO_USINT(PAR_WarnFuelLevel_Low);
send_data384[1]:=UINT_TO_USINT(PAR_WarnHydOilTem_High);
send_data384[2]:=UINT_TO_USINT(PAR_WarnOilPress_Low);
send_data384[3]:=UINT_TO_USINT(PAR_WarnWaterTem_High);
send_data384[4]:=UINT_TO_USINT(PAR_HydOilPress_PosFull MOD 256);
send_data384[5]:=UINT_TO_USINT(PAR_HydOilPress_PosFull/256);
send_data384[6]:=UINT_TO_USINT(PAR_HydOilPress_NegFull MOD 256);
send_data384[7]:=UINT_TO_USINT(PAR_HydOilPress_NegFull/256);
CAN1_SEND_384(xEnable:= TIME_1000ms.Q, eChannel:= 0, udiID:= 16#384, xExtended:=FALSE, usiDLC:=8 , aData:=send_data384);

send_data484[0]:=UINT_TO_USINT(PAR_HydOilPilotPress_PosFull MOD 256);
send_data484[1]:=UINT_TO_USINT(PAR_HydOilPilotPress_PosFull/256);
send_data484[2]:=UINT_TO_USINT(PAR_HydOilPilotPress_NegFull MOD 256);
send_data484[3]:=UINT_TO_USINT(PAR_HydOilPilotPress_NegFull/256);
send_data484[4]:=UINT_TO_USINT(PAR_TensionSensor_PosFull MOD 256);
send_data484[5]:=UINT_TO_USINT(PAR_TensionSensor_PosFull/256);
send_data484[6]:=UINT_TO_USINT(PAR_TensionSensor_NegFull MOD 256);
send_data484[7]:=UINT_TO_USINT(PAR_TensionSensor_NegFull/256);
CAN1_SEND_484(xEnable:= TIME_1000ms.Q, eChannel:= 0, udiID:= 16#484, xExtended:=FALSE, usiDLC:=8 , aData:=send_data484);

send_data584[0]:=UINT_TO_USINT(PAR_TensionSensor_Range MOD 256);
send_data584[1]:=UINT_TO_USINT(PAR_TensionSensor_Range/256);


IF  CANI_IB_VAR34_BOOL AND CANI_IB_VAR18E1 THEN 
	temp_bool1:=TRUE;
ELSE
	temp_bool1:=FALSE;
END_IF
tp_20s(IN:=temp_bool1,PT:=T#30S);

IF 	tp_20s.Q THEN
	send_data584[2]:=UINT_TO_USINT(PAR_ValveC_PosFull MOD 256);
	send_data584[3]:=UINT_TO_USINT(PAR_ValveC_PosFull/256);
	send_data584[4]:=UINT_TO_USINT(PAR_ValveC_NegFull MOD 256);
	send_data584[5]:=UINT_TO_USINT(PAR_ValveC_NegFull/256);
ELSE
	send_data584[2]:=UINT_TO_USINT(PWM_Y39 MOD 256);
	send_data584[3]:=UINT_TO_USINT(PWM_Y39/256);
	send_data584[4]:=UINT_TO_USINT(PWM_Y40 MOD 256);
	send_data584[5]:=UINT_TO_USINT(PWM_Y40/256);
END_IF
(*send_data584[6]:=UINT_TO_USINT(PWM_Y41 MOD 256);
send_data584[7]:=UINT_TO_USINT(PWM_Y41/256);*)
send_data584[6]:=UINT_TO_USINT(PAR_ValveD_PosFull MOD 256);
send_data584[7]:=UINT_TO_USINT(PAR_ValveD_PosFull/256);
CAN1_SEND_584(xEnable:= TIME_1000ms.Q, eChannel:= 0, udiID:= 16#584, xExtended:=FALSE, usiDLC:=8 , aData:=send_data584);

(*send_data684[0]:=UINT_TO_USINT(PWM_Y42 MOD 256);
send_data684[1]:=UINT_TO_USINT(PWM_Y42/256);*)
send_data684[0]:=UINT_TO_USINT(PAR_ValveD_NegFull MOD 256);
send_data684[1]:=UINT_TO_USINT(PAR_ValveD_NegFull/256);
send_data684[2]:=BYTE_TO_USINT(PAR_MainPumpChioce);
send_data684[3]:=BYTE_TO_USINT(PAR_M4ValveChioce);
send_data684[4]:=BYTE_TO_USINT(PAR_MotorChioce);
send_data684[5]:=UINT_TO_BYTE(PAR_KP);
send_data684[6]:=(PAR_KI);
send_data684[7]:=(PAR_KD);

CAN1_SEND_684(xEnable:= TIME_1000ms.Q, eChannel:= 0, udiID:= 16#684, xExtended:=FALSE, usiDLC:=8 , aData:=send_data684);

send_data784[0]:=UINT_TO_USINT(CANO_MainWinchTension MOD 256);
send_data784[1]:=UINT_TO_USINT(CANO_MainWinchTension/256);
send_data784[2]:=UINT_TO_USINT(CANO_LoadRate MOD 256);
send_data784[3]:=UINT_TO_USINT(CANO_LoadRate/256);
send_data784[4]:=UINT_TO_USINT(0 MOD 256);
send_data784[5]:=UINT_TO_USINT(0/256);
send_data784[6]:=PACK(B0:=JINZHI_LIGHT,B1:=ZAISHENG_LIGHT,B2:=GAOPAIWEN_LIGHT,B3:=DEF_LIGHT  OR JIASHIYUANWARN_LIGHT ,
					  B4:=0,B5:=0,B6:=0,B7:=0);
send_data784[7]:=urea_level;
CAN1_SEND_784(xEnable:= TIME_200ms.Q, eChannel:= 0, udiID:= 16#784, xExtended:=FALSE, usiDLC:=8 , aData:=send_data784);

send_data586[0]:=UINT_TO_USINT(PAR_MainWinchLaLi_Low MOD 256);
send_data586[1]:=UINT_TO_USINT(PAR_MainWinchLaLi_Low/256);
send_data586[2]:=UINT_TO_USINT(0 MOD 256);
send_data586[3]:=UINT_TO_USINT(0/256);
send_data586[4]:=UINT_TO_USINT(0 MOD 256);
send_data586[5]:=UINT_TO_USINT(0/256);
send_data586[6]:=UINT_TO_USINT(0 MOD 256);
send_data586[7]:=UINT_TO_USINT(0/256);
CAN1_SEND_586(xEnable:= TIME_1000ms.Q, eChannel:= 0, udiID:= 16#586, xExtended:=FALSE, usiDLC:=8 , aData:=send_data586);

send_data786[0]:=UINT_TO_USINT(0 MOD 256);
send_data786[1]:=UINT_TO_USINT(0/256);
send_data786[2]:=UINT_TO_USINT(0 MOD 256);
send_data786[3]:=UINT_TO_USINT(0/256);
send_data786[4]:=UINT_TO_USINT(0 MOD 256);
send_data786[5]:=UINT_TO_USINT(0/256);
send_data786[6]:=UINT_TO_USINT(0 MOD 256);
send_data786[7]:=PACK(B0:=DI_LHandle_SB1,B1:=DI_LHandle_SB2,B2:=DI_LHandle_SB3,B3:=DI_LHandle_SB4,
					  B4:=DI_RHandle_SB5,B5:=DI_RHandle_SB6,B6:=DI_RHandle_SB8A,B7:=DI_RHandle_SB8B);
CAN1_SEND_786(xEnable:= TIME_200ms.Q, eChannel:= 0, udiID:= 16#786, xExtended:=FALSE, usiDLC:=8 , aData:=send_data786);

send_data587[0]:=UINT_TO_USINT(PWM_Y45 MOD 256);
send_data587[1]:=UINT_TO_USINT(PWM_Y45/256);
send_data587[2]:=UINT_TO_USINT(PWM_Y46 MOD 256);
send_data587[3]:=UINT_TO_USINT(PWM_Y46/256);
send_data587[4]:=UINT_TO_USINT(0 MOD 256);
send_data587[5]:=UINT_TO_USINT(0/256);
send_data587[6]:=UINT_TO_USINT(GVL_SaveEngine.SaveEngineMode MOD 256);//UINT_TO_USINT(0 MOD 256);
send_data587[7]:=UINT_TO_USINT(GVL_SaveEngine.SaveEngineMode/256);//UINT_TO_USINT(0/256);
CAN1_SEND_587(xEnable:= TIME_1000ms.Q, eChannel:= 0, udiID:= 16#587, xExtended:=FALSE, usiDLC:=8 , aData:=send_data587);

send_data687[0]:=UINT_TO_USINT(PWM_Y49 MOD 256);
send_data687[1]:=UINT_TO_USINT(PWM_Y49/256);
send_data687[2]:=UINT_TO_USINT(PWM_Y60 MOD 256);
send_data687[3]:=UINT_TO_USINT(PWM_Y60/256);
send_data687[4]:=UINT_TO_USINT(PWM_Y61 MOD 256);
send_data687[5]:=UINT_TO_USINT(PWM_Y61/256);
send_data687[6]:=UINT_TO_USINT(CANI_JOYX_L MOD 256);
send_data687[7]:=UINT_TO_USINT(CANI_JOYX_L/256);
//CAN1_SEND_687(xEnable:= TIME_1000ms.Q, eChannel:= 0, udiID:= 16#687, xExtended:=FALSE, usiDLC:=8 , aData:=send_data687);
CAN1_SEND_687(xEnable:= TIME_100ms.Q, eChannel:= 0, udiID:= 16#687, xExtended:=FALSE, usiDLC:=8 , aData:=send_data687);


send_data787[0]:=PACK(B0:=0,B1:=0,B2:=DOH_Y50,B3:=DOH_Y51,
					  B4:=DOH_Y52,B5:=DOH_Y53,B6:=DOH_Y54,B7:=DOH_Y55);
send_data787[1]:=PACK(B0:=DOH_Y56,B1:=DOH_Y57,B2:=DOH_Y58,B3:=DOH_JK1,
					  B4:=DOH_JK2,B5:=DOH_JK3,B6:=DOH_JK4,B7:=DOH_70);
send_data787[2]:=PACK(B0:=DOH_73,B1:=DOH_B1,B2:=0,B3:=0,
					  B4:=Y71OutPutState,B5:=Y72OutPutState,B6:=Y73,B7:=0);//0改为Y71 72 73 
send_data787[3]:=UINT_TO_USINT(0);
send_data787[4]:=UINT_TO_USINT(CANI_JOYY_L MOD 256);
send_data787[5]:=UINT_TO_USINT(CANI_JOYY_L/256);
send_data787[6]:=UINT_TO_USINT(CANI_JOYX_R MOD 256);
send_data787[7]:=UINT_TO_USINT(CANI_JOYX_R/256);
//CAN1_SEND_787(xEnable:= TIME_1000ms.Q, eChannel:= 0, udiID:= 16#787, xExtended:=FALSE, usiDLC:=8 , aData:=send_data787);
CAN1_SEND_787(xEnable:= TRUE, eChannel:= 0, udiID:= 16#787, xExtended:=FALSE, usiDLC:=8 , aData:=send_data787);

send_data381[0]:=UINT_TO_USINT(PAR_Valve2_NegFull MOD 256);
send_data381[1]:=UINT_TO_USINT(PAR_Valve2_NegFull/256);
send_data381[2]:=UINT_TO_USINT(PAR_Valve3_PosFull MOD 256);
send_data381[3]:=UINT_TO_USINT(PAR_Valve3_PosFull/256);
send_data381[4]:=UINT_TO_USINT(PAR_Valve3_NegFull MOD 256);
send_data381[5]:=UINT_TO_USINT(PAR_Valve3_NegFull/256);
send_data381[6]:=UINT_TO_USINT(CANO_MainPUMP_Press1 MOD 256);
send_data381[7]:=UINT_TO_USINT(CANO_MainPUMP_Press1/256);
CAN1_SEND_381(xEnable:= TIME_200ms.Q, eChannel:= 0, udiID:= 16#381, xExtended:=FALSE, usiDLC:=8 , aData:=send_data381);

send_data481[0]:=UINT_TO_USINT(PAR_Y2_NegFull MOD 256);
send_data481[1]:=UINT_TO_USINT(PAR_Y2_NegFull/256);
send_data481[2]:=UINT_TO_USINT(PAR_Valve1_PosFull MOD 256);
send_data481[3]:=UINT_TO_USINT(PAR_Valve1_PosFull/256);
send_data481[4]:=UINT_TO_USINT(PAR_Valve1_NegFull MOD 256);
send_data481[5]:=UINT_TO_USINT(PAR_Valve1_NegFull/256);
send_data481[6]:=UINT_TO_USINT(PAR_Valve2_PosFull MOD 256);
send_data481[7]:=UINT_TO_USINT(PAR_Valve2_PosFull/256);
CAN1_SEND_481(xEnable:= TIME_1000ms.Q, eChannel:= 0, udiID:= 16#481, xExtended:=FALSE, usiDLC:=8 , aData:=send_data481);

send_data781[0]:=UINT_TO_USINT(CANI_JOYY_R MOD 256);
send_data781[1]:=UINT_TO_USINT(CANI_JOYY_R/256);
send_data781[2]:=UINT_TO_USINT(PAR_Y1_PosFull MOD 256);
send_data781[3]:=UINT_TO_USINT(PAR_Y1_PosFull/256);
send_data781[4]:=UINT_TO_USINT(PAR_Y1_NegFull MOD 256);
send_data781[5]:=UINT_TO_USINT(PAR_Y1_NegFull/256);
send_data781[6]:=UINT_TO_USINT(PAR_Y2_PosFull MOD 256);
send_data781[7]:=UINT_TO_USINT(PAR_Y2_PosFull/256);
CAN1_SEND_781(xEnable:= TIME_1000ms.Q, eChannel:= 0, udiID:= 16#781, xExtended:=FALSE, usiDLC:=8 , aData:=send_data781);

send_data182[0]:=UINT_TO_USINT(CANO_MainPUMP_Press2 MOD 256);
send_data182[1]:=UINT_TO_USINT(CANO_MainPUMP_Press2/256);
send_data182[2]:=UINT_TO_USINT(CANO_Fubeng_Press MOD 256);
send_data182[3]:=UINT_TO_USINT(CANO_Fubeng_Press/256);
send_data182[4]:=UINT_TO_USINT(AI_P11 MOD 256);
send_data182[5]:=UINT_TO_USINT(AI_P11/256);
send_data182[6]:=UINT_TO_USINT(AI_P12 MOD 256);
send_data182[7]:=UINT_TO_USINT(AI_P12/256);
CAN1_SEND_182(xEnable:= TIME_200ms.Q, eChannel:= 0, udiID:= 16#182, xExtended:=FALSE, usiDLC:=8 , aData:=send_data182);

send_data183[0]:=UINT_TO_USINT(AI_P6 MOD 256);
send_data183[1]:=UINT_TO_USINT(AI_P6/256);
send_data183[2]:=UINT_TO_USINT(PWM_Y41 MOD 256);
send_data183[3]:=UINT_TO_USINT(PWM_Y41/256);
send_data183[4]:=UINT_TO_USINT(PWM_Y42 MOD 256);
send_data183[5]:=UINT_TO_USINT(PWM_Y42/256);
send_data183[6]:=UINT_TO_USINT(PWM_Y63 MOD 256);
send_data183[7]:=UINT_TO_USINT(PWM_Y63/256);
CAN1_SEND_183(xEnable:= TIME_200ms.Q, eChannel:= 0, udiID:= 16#183, xExtended:=FALSE, usiDLC:=8 , aData:=send_data183);


send_data283[0]:=UINT_TO_USINT(CANI_JOY_Jiao_L MOD 256);
send_data283[1]:=UINT_TO_USINT(CANI_JOY_Jiao_L/256);
send_data283[2]:=UINT_TO_USINT(CANI_JOY_Jiao_R MOD 256);
send_data283[3]:=UINT_TO_USINT(CANI_JOY_Jiao_R/256);
send_data283[4]:=UINT_TO_USINT(0 MOD 256);
send_data283[5]:=UINT_TO_USINT(0/256);
send_data283[6]:=UINT_TO_USINT(0 MOD 256);
send_data283[7]:=UINT_TO_USINT(0/256);
CAN1_SEND_283(xEnable:= TIME_200ms.Q, eChannel:= 0, udiID:= 16#283, xExtended:=FALSE, usiDLC:=8 , aData:=send_data283);

send_data18F00001[0]:=UINT_TO_USINT(GVL_SaveEngine.AI_PAtomsPre MOD 256);//蓄能器气压
send_data18F00001[1]:=UINT_TO_USINT(GVL_SaveEngine.AI_PAtomsPre/256);
send_data18F00001[2]:=UINT_TO_USINT(GVL_SaveEngine.AI_PAcPre MOD 256);//蓄能器油压
send_data18F00001[3]:=UINT_TO_USINT(GVL_SaveEngine.AI_PAcPre/256);
send_data18F00001[4]:=UINT_TO_USINT(GVL_SaveEngine.AI_PM1Pre MOD 256);//M1压力
send_data18F00001[5]:=UINT_TO_USINT(GVL_SaveEngine.AI_PM1Pre/256);
send_data18F00001[6]:=UINT_TO_USINT(GVL_SaveEngine.AI_PM2Pre MOD 256);//M2压力
send_data18F00001[7]:=UINT_TO_USINT(GVL_SaveEngine.AI_PM2Pre/256);
//CAN1_SEND_18F00001(xEnable:= TIME_200ms.Q, eChannel:= 0, udiID:= 16#18F00001, xExtended:=TRUE, usiDLC:=8 , aData:=send_data18F00001);
CAN1_SEND_18F00001(xEnable:= TRUE, eChannel:= 0, udiID:= 16#18F00001, xExtended:=TRUE, usiDLC:=8 , aData:=send_data18F00001);

send_data18F00002[0]:=UINT_TO_USINT(GVL_SaveEngine.SaveEngineMode MOD 256);//节能模式0-5
IF SaveEngineState THEN
	send_data18F00002[1].0:=TRUE;//bit0:关，bit1:开
END_IF
IF (NOT SaveEngineState) THEN
	send_data18F00002[1].0:=0;//bit0:关，bit1:开
END_IF
IF GVL_SaveEngine.AcDecompression THEN
	send_data18F00002[1].1:=TRUE;//bit0:关，bit1:开
END_IF
IF (NOT GVL_SaveEngine.AcDecompression) THEN
	send_data18F00002[1].1:=0;//bit0:关，bit1:开
END_IF


send_data18F00002[2].0:=(GVL_SaveEngine.Y71OutPutState );//bit0:Y71：on/off,bit1:Y72：on/off
send_data18F00002[2].1:=(GVL_SaveEngine.Y72OutPutState );//bit0:Y71：on/off,bit1:Y72：on/off
send_data18F00002[2].2:=(Y73 );//bit0:Y71：on/off,bit1:Y72：on/off,bit2:Y73：on/off
IF (GVL_SaveEngine.AI_PAtomsPre<165) THEN//bit0:气压低报警
	send_data18F00002[3].0:=1;
ELSE
	send_data18F00002[3].0:=0;
END_IF
//bit1:蓄能器气压传感器报警
	send_data18F00002[3].1:=CANO_SensorError_PAtomsPre;
//bit2:蓄能器油压传感器报警
	send_data18F00002[3].2:=CANO_SensorError_PAcPre;
//bit3:M1压力传感器报警
	send_data18F00002[3].3:=CANO_SensorError_PM1;
//bit4:M2压力传感器报警
	send_data18F00002[3].4:=CANO_SensorError_PM2;
	
	send_data18F00002[4]:=UINT_TO_USINT(REAL_TO_UINT(Max_MainWinchTension) MOD 256);
	send_data18F00002[5]:=UINT_TO_USINT(REAL_TO_UINT(Max_MainWinchTension) / 256);
//CAN1_SEND_18F00002(xEnable:= TIME_200ms.Q, eChannel:= 0, udiID:= 16#18F00002, xExtended:=TRUE, usiDLC:=8 , aData:=send_data18F00002);
CAN1_SEND_18F00002(xEnable:= TRUE, eChannel:= 0, udiID:= 16#18F00002, xExtended:=TRUE, usiDLC:=8 , aData:=send_data18F00002);






CAN1RECEIVE_101(xEnable:=TRUE , eChannel:= 0, xExtended:= FALSE, aData=> receive_data101, udiID:= 16#101);
//临时解锁动态码
IF(receive_data101[1]=16#11)THEN
	swGpsPrivate.caculateCodeH(code1:=CANO_engine_hour_h,code2:=TO_DINT(CANO_engine_hour_m),result =>CANO_DONGTAIMA1);
	swGpsPrivate.caculateCodeL(code1:=CANO_engine_hour_h,code2:=TO_DINT(CANO_engine_hour_m),result =>CANO_DONGTAIMA2);
	send_data102[0]:=receive_data101[0];
	send_data102[1]:=16#11;
	send_data102[2]:=DINT_TO_BYTE((CANO_DONGTAIMA1 MOD 65536) MOD 256);
	send_data102[3]:=DINT_TO_BYTE((CANO_DONGTAIMA1 MOD 65536)/256);
	send_data102[4]:=DINT_TO_BYTE((CANO_DONGTAIMA1 / 65536) MOD 256);
	send_data102[5]:=DINT_TO_BYTE((CANO_DONGTAIMA2 MOD 65536) MOD 256);
	send_data102[6]:=DINT_TO_BYTE((CANO_DONGTAIMA2 MOD 65536)/256);
	send_data102[7]:=DINT_TO_BYTE((CANO_DONGTAIMA2 / 65536) MOD 256);
	IF tCounter<500 THEN
		tCounter:=tCounter+1;
		CAN1_SEND_102(xEnable:= TRUE, eChannel:= 0, udiID:= 16#102, xExtended:=FALSE, usiDLC:=8 , aData:=send_data102);
	ELSE
		receive_data101[1]:=0;
	END_IF
END_IF
swGpsPrivate.swEmergentUnlock(PH:=CANO_DONGTAIMA1,PL:=CANO_DONGTAIMA2,result=>VarGpsTempUnlockPassword2);

//永久解锁动态码
IF(receive_data101[1]=16#21)THEN
	swGpsPrivate.caculateCodeH(code1:=CANO_engine_hour_h,code2:=TO_DINT(CANO_engine_hour_m),result =>CANO_DONGTAIMA1);
	swGpsPrivate.caculateCodeL(code1:=x1,code2:=x2,result =>CANO_DONGTAIMA2);
	send_data102[0]:=receive_data101[0];
	send_data102[1]:=16#21;
	send_data102[2]:=DINT_TO_BYTE((CANO_DONGTAIMA1 MOD 65536) MOD 256);
	send_data102[3]:=DINT_TO_BYTE((CANO_DONGTAIMA1 MOD 65536)/256);
	send_data102[4]:=DINT_TO_BYTE((CANO_DONGTAIMA1 / 65536) MOD 256);
	send_data102[5]:=DINT_TO_BYTE((CANO_DONGTAIMA2 MOD 65536) MOD 256);
	send_data102[6]:=DINT_TO_BYTE((CANO_DONGTAIMA2 MOD 65536)/256);
	send_data102[7]:=DINT_TO_BYTE((CANO_DONGTAIMA2 / 65536) MOD 256);
	IF tCounter<500 THEN
		tCounter:=tCounter+1;
		CAN1_SEND_102(xEnable:= TRUE, eChannel:= 0, udiID:= 16#102, xExtended:=FALSE, usiDLC:=8 , aData:=send_data102);
	ELSE
		receive_data101[1]:=0;
	END_IF
END_IF
IF(receive_data101[1]=0)THEN
	tCounter:=0;
END_IF
swGpsPrivate.swGpsPermanentCancel(PH:=CANO_DONGTAIMA1,PL:=CANO_DONGTAIMA2,result=>VarGpsYongJiuUnlockPassword2);

END_PROGRAM

